// Condition to request disable send
      A #s_OPO98_Dispatch;// Correcting of the item is completed
      O #s_Request_Merge_Action;// Merge action is requested
      O #s_Transfer_Sort_Active;// Sorting a carrier is active
      O #s_Transfer_Merge_Active;
      O(;// When carrier at TRS01 is for OPO and TRS05 is not ready to receive an item
      A #t_TRS01_Item_Req_Sort;
      AN #s_TRS05_Ready_To_Receive;// TRS05 contain an item or not RTR
      );
      O #t_TRS05_Item_For_Merge;// Item is ready to be merged at the induct position
      O #s_TRS02_Req_Dis_Send;// Sorting is required for an item with valid LNK
      O #s_Merge_Act_Prst_PEC_Occ;// Merge action is active and the present PEC is still occupied
      = #t_TRS01_Ext_Req_Dis_Send;

      CALL #s_TRS01_FB_EQP_Basic
      (  i_ID_Section                := #i_TRS01_ID ,
         i_Basic_Offset              := #i_TRS01_Setting.Basic.Offset ,
         i_DB_PLT                    := #i_TRS01_DB_PLT ,
         i_DB_PLT_DwnStr             := #i_TRS02_DB_PLT ,
         i_DB_Event                  := "DB_Event_Section" ,
         i_Conveyor_Speed            := #s_TRS01_Selected_Speed ,
         i_Run_Out_Distance          := #s_TRS01_Selected_Run_Out ,
         i_Start_Up_Distance         := #s_TRS01_Selected_Startup ,
         i_Minimum_Gap               := #i_TRS01_Setting.Basic.Minimum_Gap ,
         i_Add_Gap_Stop              := #i_TRS01_Setting.Basic.Add_Gap_Stop ,
         i_Minimum_H2H               := #i_TRS01_Setting.Basic.Minimum_H2H ,
         i_Add_H2H_Stop              := #i_TRS01_Setting.Basic.Add_H2H_Stop ,
         i_CFG_Cascade_Delay_Time    := 30 ,
         i_CFG_Strt_Up_T_E_Save      := "DB_Setting".common.Start_Up_Time_E_Save ,
         i_CFG_Run_Out_E_Save        := "DB_Setting".common.Run_Out_Time_E_Save ,
         i_CFG_Stop_T_E_Save         := "DB_Setting".common.Stop_Time_E_Save ,
         i_PPI_Displacement          := 0 ,
         i_Dwnstr_PLT_Pos            := #s_TRS01_EOS_PEC_Pos ,
         i_CFG_Disbl_E_Save          := "DB_Setting".common.Disable_Energy_Saving ,
         i_CFG_Slave_Mode            := FALSE ,
         i_CFG_Del_Window_Codes      := FALSE ,
         i_Available_IO              := #i_IO_Available ,
         i_Safety_OK                 := #i_Safety_OK ,
         i_CMD_Enable                := #i_CMD_Enable ,
         i_CMD_Start                 := #i_CMD_Start ,
         i_Ext_Req_Stop              := #s_TRS01_Ext_Req_Stop ,
         i_Ext_Req_Halt              := FALSE ,
         i_Ext_Req_Dis_Send          := #t_TRS01_Ext_Req_Dis_Send ,
         i_Ext_Req_Rst_ESave         := FALSE ,
         i_OS_Direction_Change       := FALSE ,
         i_Clr_PLT_Data              := #s_TRS01_ST_LMS_Not_Auto ,
         o_External                  := #o_TRS01_Ext_Outputs ,
         o_Motor_Run                 := #s_TRS01_Motor_Run ,
         o_ST_Items                  := #o_TRS01_ST_Items ,
         o_ST_Running                := #o_TRS01_ST_Running ,
         o_ST_Started                := #o_TRS01_ST_Started ,
         o_ST_Request_Halt           := #o_TRS01_ST_Req_Halt ,
         o_ST_Request_Stop           := #o_TRS01_ST_Req_Stop ,
         o_ST_External_Stop          := #o_TRS01_ST_Ext_Stop ,
         o_Ready_To_Restart          := #s_TRS01_Ready_To_Restart
      );

      CALL #s_TRS01_FB_TRK_Track_EOS
      (  i_Setting                   := #i_TRS01_Setting.Tracking ,
         i_DB_PLT                    := #i_TRS01_DB_PLT ,
         i_Event_DB                  := "DB_Event_Section" ,
         i_Position_PEC_Update       := #s_TRS01_EOS_PEC_Pos ,
         i_LPOS                      := #s_TRS01_EOS_PEC_LPOS ,
         i_Length_Dif_Accepted       := 0 ,
         i_CFG_Num_Missing_Error     := 3 ,
         i_CFG_Upd_Perf_WN_Level     := 80 ,
         i_CFG_Weighing_Factor       := 10 ,
         i_CFG_Default_Record        := #i_CFG_Default_Record ,
         i_Trigger_Send_Stat         := #i_Send_Statistics ,
         i_CMD_Reset                 := #i_CMD_Reset ,
         i_CFG_Clear_Double_Data     := TRUE ,
         i_OS_Direction_Change       := FALSE ,
         i_HW_MTR_Not_Auto           := #s_TRS01_ST_LMS_Not_Auto ,
         o_ST_PEC_Miss               := #s_TRS01_ST_EOS_PEC_Miss ,
         o_ST_PEC_BadTrack           := #o_TRS01_ST_EOS_PEC_BadTr
      );

      AN "M_Hardware_PN";
      JCN HA01;

      CALL #s_TRS01_FB_HW_MltSpd_LMS
      (  i_CMD_Send_Stat             := #i_Send_Statistics ,
         i_DB_PLT                    := #i_TRS01_DB_PLT ,
         i_Event_DB                  := "DB_Event_Section" ,
         i_Speed1                    := #i_TRS01_Setting.Hardware.Speed1 ,
         i_Speed1_Run_Out_Dist       := #i_TRS01_Setting.Hardware.Speed1_Run_Out_Dist ,
         i_Speed1_Start_Up_Dist      := #i_TRS01_Setting.Hardware.Speed1_Start_Up_Dist ,
         i_CFG_Motor_Switch_Time     := 0 ,
         i_CMD_Select_Speed          := 1 ,
         i_Available_IO              := #i_IO_Available ,
         i_LMS_NotPrsnt              := #i_TRS01_LMS_Not_Prsnt ,
         i_LMS_Error                 := #i_TRS01_LMS_Error ,
         i_IO_LMS_Auto               := #i_TRS01_IO_LMS_Auto ,
         i_IO_LMS_Healthy            := #i_TRS01_IO_LMS_Healthy ,
         i_CMD_Reset                 := #i_CMD_Reset ,
         i_CMD_Req_Motor_Run         := #s_TRS01_Motor_Run ,
         o_IO_MTR_Fwd                := #o_TRS01_IO_MTR_Fwd ,
         o_IO_MTR_Rev                := #o_TRS01_IO_MTR_Rev ,
         o_IO_Speed_Select1          := #o_TRS01_IO_Speed_Select1 ,
         o_IO_Speed_Select2          := #o_TRS01_IO_Speed_Select2 ,
         o_ST_ASI_NotPrsnt           := #s_TRS01_ST_LMS_Not_Prsnt ,
         o_ST_ASI_Err                := #s_TRS01_ST_LMS_Error ,
         o_ST_LMS_Not_Auto           := #s_TRS01_ST_LMS_Not_Auto ,
         o_ST_LMS_Not_Hthy           := #s_TRS01_ST_LMS_Not_Hthy ,
         o_Select_Conveyor_Speed     := #s_TRS01_Selected_Speed ,
         o_Select_Run_Out_Dist       := #s_TRS01_Selected_Run_Out ,
         o_Select_Started_Up_Dist    := #s_TRS01_Selected_Startup
      );

      JU HA02;

HA01:      CALL #s_TRS01_FB_HW_MTR_PN_LMS
      (  i_CMD_Send_Stat             := #i_Send_Statistics ,
         i_DB_PLT                    := #i_TRS01_DB_PLT ,
         i_Event_DB                  := "DB_Event_Section" ,
         i_Speed                     := #i_TRS01_Setting.Hardware.Speed1 ,
         i_Run_Out_Dist              := #i_TRS01_Setting.Hardware.Speed1_Run_Out_Dist ,
         i_Start_Up_Dist             := #i_TRS01_Setting.Hardware.Speed1_Start_Up_Dist ,
         i_CFG_Motor_Switch_Time     := 0 ,
         i_CFG_In_Hardw_ID           := #i_TRS01_CFG_LMS_In_Hardw_ID ,
         i_CFG_Out_Hardw_ID          := #i_TRS01_CFG_LMS_Out_Hardw_ID ,
         i_Available_IO              := #i_IO_Available ,
         i_CMD_Reset                 := #i_CMD_Reset ,
         i_CMD_Req_Motor_Run         := #s_TRS01_Motor_Run ,
         o_ST_FieldB_NotPrsnt        := #s_TRS01_ST_LMS_Not_Prsnt ,
         o_ST_FieldB_Error           := #s_TRS01_ST_LMS_Error ,
         o_ST_LMS_Not_Auto           := #s_TRS01_ST_LMS_Not_Auto ,
         o_ST_LMS_Not_Hthy           := #s_TRS01_ST_LMS_Not_Hthy ,
         o_Select_Conveyor_Speed     := #s_TRS01_Selected_Speed ,
         o_Select_Run_Out_Dist       := #s_TRS01_Selected_Run_Out ,
         o_Select_Started_Up_Dist    := #s_TRS01_Selected_Startup
      );

HA02:      NOP 0;

      CALL #s_TRS01_FB_DAT_T
      (  i_ID                        := #i_TRS01_ID ,
         i_DB_Event                  := "DB_Event_Section" ,
         i_DB_PLT_Lost_And_Found     := #i_DB_PLT_Lost_And_Found ,
         i_DB_Send_FIFO_PNPN         := #i_DB_Send_FIFO_PNPN
      );

      CALL #s_TRS01_FB_DAT
      (  i_ID_Section                := #i_TRS01_ID ,
         i_DB_Event                  := "DB_Event_Section" ,
         i_PLC_Log_FIFO_DB           := "DB_LOG_Event_FIFO" ,
         i_CFG_BPI_Log_Level         := "DB_Setting".common.External_Log_Level ,
         i_CFG_PLC_Log_Level         := "DB_Setting".common.Internal_Log_Level ,
         i_CFG_PLC_Log_Route_Msgs    := FALSE ,
         i_CFG_PLC_LOG_BPI_Stat      := FALSE
      );

NETWORK
TITLE = IA: Transport section TRS02
      NOP 0;

// Condition to request stop
      A #s_TRS02_ST_LMS_Not_Prsnt;// LMS and PEC related errors
      O #s_TRS02_ST_LMS_Error;
      O #s_TRS02_ST_LMS_Not_Auto;
      O #s_TRS02_ST_LMS_Not_Hthy;
      O(;// SWS, MSO and TRS04 errors considered-
      A #s_SWS03_STM_Err;// when sorting is required for an item
      A #s_Sorting_Required;
      );
      O #s_TRS04_ST_Prsnt_PEC_Blk;// Present PEC blockage shall stop TRS02 at all times
      O(;// ASi slave errors of HAC PEC
      O #s_TRS04_ST_FieldB_Not_Prsnt;
      O #s_TRS04_ST_FieldB_Error;
      A #i_IO_Available;
      );
      = #s_TRS02_Ext_Req_Stop;

// Condition to request halt
      AN #s_SWS03_Req_Down;// Whenever SWS is requested to go down
      O(;
      A #s_TRS02_Carr_In_Pos;// When carrier is in position, sorting is required
      A #s_Sorting_Required;
      );
      O(;// Consider SWS related errors if not in down position
      A #s_SWS03_ST_LMS_Not_Prsnt;
      O #s_SWS03_ST_LMS_Error;
      O #s_SWS03_ST_LMS_Not_Auto;
      O #s_SWS03_ST_LMS_Not_Hthy;
      O #s_SWS03_ST_Move_TimeOut;
      O #s_SWS03_ST_PS_Double;
      AN #s_SWS03_ST_Down;
      );
      O(;// Consider MSO related errors if not in down position
      A #s_MSO99_ST_LMS_Not_Prsnt;
      O #s_MSO99_ST_LMS_Error;
      O #s_MSO99_ST_LMS_Not_Auto;
      O #s_MSO99_ST_LMS_Not_Hthy;
      O #s_MSO99_ST_Move_TimeOut;
      O #s_MSO99_ST_PS_Double;
      AN #s_MSO99_ST_Down;
      );
      O(;// When merge action is active, SWS is down
      A #s_Transfer_Merge_Active;// and the downstream is not RTR
      AN #t_TRS02_Dwnstr_RTR;
      A #i_SWS03_IO_PS_Down;
      );
      O #s_TRS04_ST_HAC_PEC_Blk;// ASi slave and PEC errors of HAC PEC
      O #s_TRS04_ST_FieldB_Not_Prsnt;
      O #s_TRS04_ST_FieldB_Error;
      O #s_TRS04_ST_SOS_PEC_Blk;// ASi slave and PEC errors of TRS04
      ON #s_TRS04_IO_Available_LMS;
      O(;// Latch the halt if stopped while merge is active
      A #s_Transfer_Merge_Active;
      O #s_TRS02_Ext_Req_Halt;
      A #i_CMD_Controlled_Stop;
      );
      O #s_Transfer_Merge_Active;// When merge action is active
      = #s_TRS02_Ext_Req_Halt;

// Condition to disable send
      A #i_CMD_Controlled_Stop;
      = #s_TRS02_Ext_Req_Dis_Send;

// Condition to reset Esave
      AN #i_TRS04_IO_NOT_Prsnt_PEC;
      = #t_TRS02_Ext_Req_Rst_Esav;

      CALL #s_TRS02_FB_EQP_Basic
      (  i_ID_Section                := #i_TRS02_ID ,
         i_Basic_Offset              := #i_TRS02_Setting.Basic.Offset ,
         i_DB_PLT                    := #i_TRS02_DB_PLT ,
         i_DB_PLT_DwnStr             := #i_DB_PLT_Dwnstr ,
         i_DB_Event                  := "DB_Event_Section" ,
         i_Conveyor_Speed            := #s_TRS02_Selected_Speed ,
         i_Run_Out_Distance          := #s_TRS02_Selected_Run_Out ,
         i_Start_Up_Distance         := #s_TRS02_Selected_Startup ,
         i_Minimum_Gap               := #i_TRS02_Setting.Basic.Minimum_Gap ,
         i_Add_Gap_Stop              := #i_TRS02_Setting.Basic.Add_Gap_Stop ,
         i_Minimum_H2H               := #i_TRS02_Setting.Basic.Minimum_H2H ,
         i_Add_H2H_Stop              := #i_TRS02_Setting.Basic.Add_H2H_Stop ,
         i_CFG_Dieback_Position      := #t_TRS02_CFG_MSO_Pos ,
         i_CFG_Cascade_Delay_Time    := 0 ,
         i_CFG_Strt_Up_T_E_Save      := "DB_Setting".common.Start_Up_Time_E_Save ,
         i_CFG_Run_Out_E_Save        := "DB_Setting".common.Run_Out_Time_E_Save ,
         i_CFG_Stop_T_E_Save         := "DB_Setting".common.Stop_Time_E_Save ,
         i_PPI_Displacement          := 0 ,
         i_Dwnstr_PLT_Pos            := #s_TRS04_SOS_PEC_Pos ,
         i_CFG_Disbl_E_Save          := "DB_Setting".common.Disable_Energy_Saving ,
         i_CFG_Slave_Mode            := FALSE ,
         i_CFG_Del_Window_Codes      := FALSE ,
         i_Available_IO              := #i_IO_Available ,
         i_Safety_OK                 := #i_Safety_OK ,
         i_CMD_Enable                := #i_CMD_Enable ,
         i_CMD_Start                 := #i_CMD_Start ,
         i_Ext_Req_Stop              := #s_TRS02_Ext_Req_Stop ,
         i_Ext_Req_Halt              := #s_TRS02_Ext_Req_Halt ,
         i_Ext_Req_Dis_Send          := #s_TRS02_Ext_Req_Dis_Send ,
         i_Ext_Req_Rst_ESave         := #t_TRS02_Ext_Req_Rst_Esav ,
         i_OS_Direction_Change       := FALSE ,
         i_Clr_PLT_Data              := FALSE ,
         o_External                  := #o_TRS02_Ext_Outputs ,
         o_Motor_Run                 := #s_TRS02_Motor_Run ,
         o_ST_Items                  := #s_TRS02_ST_Items ,
         o_ST_Running                := #o_TRS02_ST_Running ,
         o_ST_Started                := #o_TRS02_ST_Started ,
         o_ST_Request_Halt           := #o_TRS02_ST_Req_Halt ,
         o_ST_Request_Stop           := #o_TRS02_ST_Req_Stop ,
         o_ST_External_Stop          := #o_TRS02_ST_Ext_Stop ,
         o_Ready_To_Restart          := #s_TRS02_Ready_To_Restart
      );

      CALL #s_TRS02_FB_TRK_No_PEC
      (  i_DB_PLT                    := #i_TRS02_DB_PLT ,
         i_Event_DB                  := "DB_Event_Section" ,
         i_HW_MTR_Not_Auto           := #s_TRS02_ST_LMS_Not_Auto
      );

// Select speed
      AN #s_TRS02_Req_2nd_Speed;
      JCN IA01;

      L 1;
      T #t_TRS02_Select_Speed;
      JU IA02;

IA01:      L 2;
      T #t_TRS02_Select_Speed;

IA02:      AN "M_Hardware_PN";
      JCN IA03;

      CALL #s_TRS02_FB_HW_MltSpd_LMS
      (  i_CMD_Send_Stat             := #i_Send_Statistics ,
         i_DB_PLT                    := #i_TRS02_DB_PLT ,
         i_Event_DB                  := "DB_Event_Section" ,
         i_Speed1                    := #i_TRS02_Setting.Hardware.Speed1 ,
         i_Speed1_Run_Out_Dist       := #i_TRS02_Setting.Hardware.Speed1_Run_Out_Dist ,
         i_Speed1_Start_Up_Dist      := #i_TRS02_Setting.Hardware.Speed1_Start_Up_Dist ,
         i_Speed2                    := #i_TRS02_Setting.Hardware.Speed2 ,
         i_Speed2_Run_Out_Dist       := #i_TRS02_Setting.Hardware.Speed2_Run_Out_Dist ,
         i_Speed2_Start_Up_Dist      := #i_TRS02_Setting.Hardware.Speed2_Start_Up_Dist ,
         i_CFG_Motor_Switch_Time     := 0 ,
         i_CMD_Select_Speed          := #t_TRS02_Select_Speed ,
         i_Available_IO              := #i_IO_Available ,
         i_LMS_NotPrsnt              := #i_TRS02_LMS_Not_Prsnt ,
         i_LMS_Error                 := #i_TRS02_LMS_Error ,
         i_IO_LMS_Auto               := #i_TRS02_IO_LMS_Auto ,
         i_IO_LMS_Healthy            := #i_TRS02_IO_LMS_Healthy ,
         i_CMD_Reset                 := #i_CMD_Reset ,
         i_CMD_Req_Motor_Run         := #s_TRS02_Motor_Run ,
         i_CMD_Req_Motor_Reverse     := FALSE ,
         o_IO_MTR_Fwd                := #o_TRS02_IO_MTR_Fwd ,
         o_IO_MTR_Rev                := #o_TRS02_IO_MTR_Rev ,
         o_IO_Speed_Select1          := #o_TRS02_IO_Speed_Select1 ,
         o_IO_Speed_Select2          := #o_TRS02_IO_Speed_Select2 ,
         o_ST_ASI_NotPrsnt           := #s_TRS02_ST_LMS_Not_Prsnt ,
         o_ST_ASI_Err                := #s_TRS02_ST_LMS_Error ,
         o_ST_LMS_Not_Auto           := #s_TRS02_ST_LMS_Not_Auto ,
         o_ST_LMS_Not_Hthy           := #s_TRS02_ST_LMS_Not_Hthy ,
         o_Select_Conveyor_Speed     := #s_TRS02_Selected_Speed ,
         o_Select_Run_Out_Dist       := #s_TRS02_Selected_Run_Out ,
         o_Select_Started_Up_Dist    := #s_TRS02_Selected_Startup
      );

      JU IA04;

// By default use speed 1
IA03:      L #i_TRS02_Setting.Hardware.Speed1;
      T #t_TRS02_Speed;
      L #i_TRS02_Setting.Hardware.Speed1_Run_Out_Dist;
      T #t_TRS02_Run_Out_Dist;
      L #i_TRS02_Setting.Hardware.Speed1_Start_Up_Dist;
      T #t_TRS02_Start_Up_Dist;

// Determine if speed 2 is selected
      L #t_TRS02_Select_Speed;
      L 2;
      ==I;
      JCN IA05;

      L #i_TRS02_Setting.Hardware.Speed2;
      T #t_TRS02_Speed;
      L #i_TRS02_Setting.Hardware.Speed2_Run_Out_Dist;
      T #t_TRS02_Run_Out_Dist;
      L #i_TRS02_Setting.Hardware.Speed2_Start_Up_Dist;
      T #t_TRS02_Start_Up_Dist;

IA05:      CALL #s_TRS02_FB_HW_MTR_PN_LMS
      (  i_CMD_Send_Stat             := #i_Send_Statistics ,
         i_DB_PLT                    := #i_TRS02_DB_PLT ,
         i_Event_DB                  := "DB_Event_Section" ,
         i_Speed                     := #t_TRS02_Speed ,
         i_Run_Out_Dist              := #t_TRS02_Run_Out_Dist ,
         i_Start_Up_Dist             := #t_TRS02_Start_Up_Dist ,
         i_CFG_In_Hardw_ID           := #i_TRS02_CFG_LMS_In_Hardw_ID ,
         i_CFG_Out_Hardw_ID          := #i_TRS02_CFG_LMS_Out_Hardw_ID ,
         i_Available_IO              := #i_IO_Available ,
         i_CMD_Reset                 := #i_CMD_Reset ,
         i_CMD_Req_Motor_Run         := #s_TRS02_Motor_Run ,
         o_ST_FieldB_NotPrsnt        := #s_TRS02_ST_LMS_Not_Prsnt ,
         o_ST_FieldB_Error           := #s_TRS02_ST_LMS_Error ,
         o_ST_LMS_Not_Auto           := #s_TRS02_ST_LMS_Not_Auto ,
         o_ST_LMS_Not_Hthy           := #s_TRS02_ST_LMS_Not_Hthy ,
         o_Select_Conveyor_Speed     := #s_TRS02_Selected_Speed ,
         o_Select_Run_Out_Dist       := #s_TRS02_Selected_Run_Out ,
         o_Select_Started_Up_Dist    := #s_TRS02_Selected_Startup
      );

IA04:      NOP 0;

      CALL #s_TRS02_FB_DAT_T
      (  i_ID                        := #i_TRS02_ID ,
         i_DB_Event                  := "DB_Event_Section" ,
         i_DB_PLT_Lost_And_Found     := #i_DB_PLT_Lost_And_Found ,
         i_DB_Send_FIFO_PNPN         := #i_DB_Send_FIFO_PNPN
      );

      CALL #s_TRS02_FB_DAT
      (  i_ID_Section                := #i_TRS02_ID ,
         i_DB_Event                  := "DB_Event_Section" ,
         i_PLC_Log_FIFO_DB           := "DB_LOG_Event_FIFO" ,
         i_CFG_BPI_Log_Level         := "DB_Setting".common.External_Log_Level ,
         i_CFG_PLC_Log_Level         := "DB_Setting".common.Internal_Log_Level ,
         i_CFG_PLC_Log_Route_Msgs    := FALSE ,
         i_CFG_PLC_LOG_BPI_Stat      := FALSE
      );

NETWORK
TITLE = JA: Switch section SWS03 (TSS)
      NOP 0;

// SWS Up   = Direction A = Motor up
// SWS Down = Direction B = Motor Down
// Section up status
      A #i_IO_Available;
      A #i_SWS03_IO_PS_Up;
      AN #i_SWS03_IO_PS_Down;
      = #s_SWS03_ST_Up;

// Section down status
      A #i_IO_Available;
      A #i_SWS03_IO_PS_Down;
      AN #i_SWS03_IO_PS_Up;
      = #s_SWS03_ST_Down;

// Check for error transfer module
      A #s_SWS03_ST_LMS_Not_Prsnt;
      O #s_SWS03_ST_LMS_Error;
      O #s_SWS03_ST_LMS_Not_Auto;
      O #s_SWS03_ST_LMS_Not_Hthy;
      O #s_SWS03_ST_Move_TimeOut;
      O #s_SWS03_ST_PS_Double;
      O #s_TRS04_ST_LMS_Not_Prsnt;
      O #s_TRS04_ST_LMS_Error;
      O #s_TRS04_ST_LMS_Not_Auto;
      O #s_TRS04_ST_LMS_Not_Hthy;
      O #s_TRS04_ST_Prsnt_PEC_Blk;
      O #s_TRS04_ST_SOS_PEC_Blk;
      O #s_TRS04_ST_SOS_PEC_Miss;
      O #s_TRS04_ST_FieldB_Not_Prsnt;
      O #s_TRS04_ST_FieldB_Error;
      O #s_TRS04_ST_HAC_PEC_Blk;
      O #s_MSO99_ST_LMS_Not_Prsnt;
      O #s_MSO99_ST_LMS_Error;
      O #s_MSO99_ST_LMS_Not_Auto;
      O #s_MSO99_ST_LMS_Not_Hthy;
      O #s_MSO99_ST_Move_TimeOut;
      O #s_MSO99_ST_PS_Double;
      = #s_SWS03_STM_Err;

// Condition to request stop
      A #s_SWS03_STM_Err;
      = #s_SWS03_Ext_Req_Stop;

// Condition to request position up while sorting
      A #t_TRS02_Stopped;
      A #s_TRS02_Carr_In_Pos;
      AN #i_CMD_Controlled_Stop;
      O #s_Transfer_Sort_Active;
      = #t_SWS03_Req_Up_Sorting;

// Item in position on lift after merge
      A #s_TRS04_ST_Items;
      A #s_TRS04_ST_Started;
      AN #s_TRS04_ST_Running;
      AN #s_TRS05_ST_Items;
      A #i_TRS04_IO_NOT_HAC_PEC;
      AN #i_TRS04_IO_NOT_Prsnt_PEC;
      = #s_Carrier_On_Lift_Merge;

// Condition to request position up while merging
      A #s_Request_Merge_Action;
      O(;
      A #s_Transfer_Merge_Active;
      AN #s_Carrier_On_Lift_Merge;
      );
      = #t_SWS03_Req_Up_Merging;

// Condition to request position down
      AN #t_SWS03_Req_Up_Merging;
      AN #t_SWS03_Req_Up_Sorting;
      O(;
      A #i_CMD_Start;
      AN #s_SWS03_ST_Down;
      AN #s_Transfer_Sort_Active;
      AN #s_Request_Merge_Action;
      AN #s_Transfer_Merge_Active;
      );
      = #s_SWS03_Req_Down;

      CALL #s_SWS03_FB_EQP_Switch
      (  i_Available_IO              := #i_IO_Available ,
         i_Safety_OK                 := #i_Safety_OK ,
         i_CMD_Enable                := #i_CMD_Enable ,
         i_CMD_Start                 := #i_CMD_Start ,
         i_CMD_Reset                 := #i_CMD_Reset ,
         i_IO_PS_A                   := #i_SWS03_IO_PS_Up ,
         i_IO_PS_B                   := #i_SWS03_IO_PS_Down ,
         i_Ext_Req_Stop              := #s_SWS03_Ext_Req_Stop ,
         i_Ext_Req_Halt              := FALSE ,
         i_Req_Dir_B                 := #s_SWS03_Req_Down ,
         i_Timeout_Dir               := #i_SWS03_Setting.Timeout_Dir ,
         o_CMD_MTR_Run               := #s_SWS03_Motor_Run ,
         o_CMD_MTR_Reverse           := #s_SWS03_Motor_Reverse ,
         o_ST_Running                := #o_SWS03_ST_Running ,
         o_ST_Started                := #o_SWS03_ST_Started ,
         o_ST_Request_Halt           := #o_SWS03_ST_Req_Halt ,
         o_ST_Request_Stop           := #o_SWS03_ST_Req_Stop ,
         o_ST_External_Stop          := #o_SWS03_ST_Ext_Stop ,
         o_ST_Movement_Time_out      := #s_SWS03_ST_Move_TimeOut ,
         o_ST_PS_Double              := #s_SWS03_ST_PS_Double ,
         o_Ready_To_Restart          := #s_SWS03_Ready_To_Restart
      );

      AN "M_Hardware_PN";
      JCN JA01;

      CALL #s_SWS03_FB_HW_MTR_2D_LMS
      (  i_CMD_Send_Stat             := #i_Send_Statistics ,
         i_Event_DB                  := "DB_Event_Section" ,
         i_CFG_Motor_Switch_Time     := 0 ,
         i_Available_IO              := #i_IO_Available ,
         i_Quick_Stop                := TRUE ,
         i_LMS_NotPrsnt              := #i_SWS03_LMS_Not_Prsnt ,
         i_LMS_Error                 := #i_SWS03_LMS_Error ,
         i_IO_LMS_Auto               := #i_SWS03_IO_LMS_Auto ,
         i_IO_LMS_Healthy            := #i_SWS03_IO_LMS_Healthy ,
         i_CMD_Reset                 := #i_CMD_Reset ,
         i_CMD_Req_Motor_Run         := #s_SWS03_Motor_Run ,
         i_CMD_Req_Motor_Reverse     := #s_SWS03_Motor_Reverse ,
         o_IO_MTR_Fwd                := #o_SWS03_IO_MTR_Up ,
         o_IO_MTR_Rev                := #o_SWS03_IO_MTR_Down ,
         o_IO_MTR_Dis_Quick_Stop     := #o_SWS03_IO_Dis_QS ,
         o_ST_ASI_NotPrsnt           := #s_SWS03_ST_LMS_Not_Prsnt ,
         o_ST_ASI_Err                := #s_SWS03_ST_LMS_Error ,
         o_ST_LMS_Not_Auto           := #s_SWS03_ST_LMS_Not_Auto ,
         o_ST_LMS_Not_Hthy           := #s_SWS03_ST_LMS_Not_Hthy
      );

      JU JA02;

JA01:      CALL #s_SWS03_FB_HW_MTR_2D_PN_LMS
      (  i_CMD_Send_Stat             := #i_Send_Statistics ,
         i_Event_DB                  := "DB_Event_Section" ,
         i_CFG_Motor_Switch_Time     := 0 ,
         i_CFG_In_Hardw_ID           := #i_SWS03_CFG_LMS_In_Hardw_ID ,
         i_CFG_Out_Hardw_ID          := #i_SWS03_CFG_LMS_Out_Hardw_ID ,
         i_Available_IO              := #i_IO_Available ,
         i_CMD_Reset                 := #i_CMD_Reset ,
         i_CMD_Req_Motor_Run         := #s_SWS03_Motor_Run ,
         i_CMD_Req_Motor_Reverse     := #s_SWS03_Motor_Reverse ,
         o_ST_FieldB_NotPrsnt        := #s_SWS03_ST_LMS_Not_Prsnt ,
         o_ST_FieldB_Error           := #s_SWS03_ST_LMS_Error ,
         o_ST_LMS_Not_Auto           := #s_SWS03_ST_LMS_Not_Auto ,
         o_ST_LMS_Not_Hthy           := #s_SWS03_ST_LMS_Not_Hthy
      );

JA02:      NOP 0;

      CALL #s_SWS03_FB_DAT_T
      (  i_ID                        := #i_SWS03_ID ,
         i_DB_Event                  := "DB_Event_Section"
      );

      CALL #s_SWS03_FB_DAT
      (  i_ID_Section                := #i_SWS03_ID ,
         i_DB_Event                  := "DB_Event_Section" ,
         i_PLC_Log_FIFO_DB           := "DB_LOG_Event_FIFO" ,
         i_CFG_BPI_Log_Level         := "DB_Setting".common.External_Log_Level ,
         i_CFG_PLC_Log_Level         := "DB_Setting".common.Internal_Log_Level ,
         i_CFG_PLC_Log_Route_Msgs    := FALSE ,
         i_CFG_PLC_LOG_BPI_Stat      := FALSE
      );

NETWORK
TITLE = KA: Activate 2nd speed TRS04
//When a leading edge is found from a configurable point on TRS04, the TRS will
//switch to the 2nd speed. This is done to reduce the impact of the carrier
//against the side guarding.
      NOP 0;

      L #i_TRS04_CFG_2nd_Spd_Pos;
      L 30;// Add 30cm extra, to also find leading edge in END PLT (Dummy PLT)
      +I;
      T #t_Search_Window;

      CALL "FC_PLT_Srch_Inf_Dwn"
      (  i_DB_PLT_Num                := #t_TRS04_DB_PLT_Num ,
         i_Position                  := #i_TRS04_CFG_2nd_Spd_Pos ,
         i_Window                    := #t_Search_Window ,
         i_Info                      := 1 ,
         o_Position                  := #t_Not_Used_Int ,
         o_Info                      := #t_Not_Used_Int ,
         o_LNK                       := #t_Fnd_Link_2nd_Speed ,
         o_DB_PLT_Num                := #t_Not_Used_Int ,
         o_Number_Items_Found        := #t_Not_Used_Int
      );

// When a link has been found, switch to 2nd speed
      L #t_Fnd_Link_2nd_Speed;
      L 0;
      >I;
      A #s_Transfer_Merge_Active;
      JCN KA01;

      L 2;
      T #t_TRS04_Select_Speed;
      JU KA99;

KA01:      L 1;
      T #t_TRS04_Select_Speed;

KA99:      NOP 0;

NETWORK
TITLE = LA: Push carrier out of HAC PEC
//Push carrier out of the HAC PEC to avoid deadlock during transfer merge
      NOP 0;

      AN #i_TRS04_IO_NOT_HAC_PEC;
      A #t_TRS04_Operational;
      A #t_TRS04_Stopped;
      A #s_SWS03_ST_Up;
      A #s_Transfer_Merge_Active;
      = #t_Push_Carr_Timer_Start;

      CALL "FC_On_Dly_T_0.1s"
      (  i_Start                     := #t_Push_Carr_Timer_Start ,
         i_Enable_Dly                := TRUE ,
         i_Time_Value                := 45 ,
         i_Current_Value             := #s_Push_Carr_Timer_CV ,
         o_Status                    := #t_Push_Carr_Timer_Done ,
         o_Current_Value             := #s_Push_Carr_Timer_CV
      );

      OPN #i_TRS05_DB_PLT;
      A #t_Push_Carr_Timer_Start;
      JCN LA99;

      CLR;
      = %DBX10.6;// Item at handover

LA99:      NOP 0;

NETWORK
TITLE = MA: Transport section TRS04 (TTS)
//Note that the SOS PEC connects to the TRS04 LMS but is located on section 02
//not TRS04. The SOS PEC therefor updates the section 02 tracking.
      NOP 0;

      CALL #s_TRS04_FB_EQP_Switch_D
      (  i_DB_PLT                    := #i_TRS04_DB_PLT ,
         i_DB_PLT_UpStr              := #i_TRS04_DB_PLT_End ,
         i_DB_PLT_DwnStr             := #i_TRS05_DB_PLT ,
         i_CMD_Reverse               := #s_Req_Reverse_TRS05 ,
         i_CFG_Cascade_Delay_FWD     := 0 ,
         i_CFG_Cascade_Delay_REV     := 0 ,
         o_OS_Direction_Change       := #s_TRS04_OS_Dir_Change ,
         o_CMD_MTR_Reverse           := #s_TRS04_Motor_Reverse ,
         o_Cascade_Delay_Time        := #t_Not_Used_Int
      );

      AN #s_TRS04_Motor_Reverse;
      = #s_TRS04_Motor_Forward;

// IO Available for SOS and present PEC
      A #i_IO_Available;
      AN #s_TRS04_ST_LMS_Not_Prsnt;
      AN #s_TRS04_ST_LMS_Error;
      = #s_TRS04_IO_Available_LMS;

// Note the SOS PEC is located on the section 02, not TRS04
      CALL #s_TRS04_FB_EQP_PEC_SOS
      (  i_Setting                   := #i_TRS04_Setting.PEC_1 ,
         i_DB_PLT                    := #i_TRS02_DB_PLT ,
         i_DB_Event                  := "DB_Event_Section" ,
         i_Dwnstr_PLT_Pos            := 0 ,
         i_CFG_Blockage_Length       := #i_CFG_Blockage_Length_L ,
         i_CFG_Delay_On_Filter       := 15 ,
         i_CFG_Delay_Off_Filter      := 0 ,
         i_CFG_Flickering_Length     := 60 ,
         i_CFG_Min_Product_Length    := 60 ,
         i_CFG_Preset_PEC_Latch      := #s_TRS04_ST_LMS_Not_Auto ,
         i_CFG_Track_Present         := TRUE ,
         i_CFG_Reset_Block_PEC_Oc    := FALSE ,
         i_IO_NOT_PEC                := #i_TRS04_IO_NOT_SOS_PEC ,
         i_Eqp_Available_IO          := #s_TRS04_IO_Available_LMS ,
         i_CMD_Reset                 := #i_CMD_Reset ,
         o_LPOS                      := #s_TRS04_SOS_PEC_LPOS ,
         o_PEC_Position              := #s_TRS04_SOS_PEC_Pos ,
         o_ST_PEC_Blk                := #s_TRS04_ST_SOS_PEC_Blk
      );

// Determine if the present PEC is occupied during a merge action
      A #s_Transfer_Merge_Active;
      AN #i_TRS04_IO_NOT_Prsnt_PEC;
      S #s_Merge_Act_Prst_PEC_Occ;

      A #i_TRS04_IO_NOT_Prsnt_PEC;
      R #s_Merge_Act_Prst_PEC_Occ;

// Selection of displacement for present PEC blockage detection
      A #s_SWS03_ST_Up;
      JCN MA01;

      L #t_TRS04_Displ;// Displacement of transfer
      JU MA02;

MA01:      L #t_TRS02_Displ;// Displacement of mainline TB
MA02:      T #t_Displ_PECT_Prst;

// Blockage length present PEC
      L #i_CFG_Blockage_Length_L;
      L "DB_Setting".Common_TTT.SBT_Length;// Additional SBT length because of the (+/-)diagonal position of present PEC
      +I;
      T #t_PECT_Prst_Blck_length;// Blockage length present PEC

      CALL #s_TRS04_FB_EQP_PECT_Prst
      (  i_CFG_Blockage_Length       := #t_PECT_Prst_Blck_length ,
         i_CFG_Delay_On_Filter       := 0 ,
         i_CFG_Reset_Block_PEC_Oc    := FALSE ,
         i_CFG_Time_Displacement     := TRUE ,
         i_IO_NOT_PEC                := #i_TRS04_IO_NOT_Prsnt_PEC ,
         i_Eqp_Available_IO          := #s_TRS04_IO_Available_LMS ,
         i_CMD_Reset                 := #i_CMD_Reset ,
         i_Displacement              := #t_Displ_PECT_Prst ,
         o_ST_PEC_Blk                := #s_TRS04_ST_Prsnt_PEC_Blk ,
         o_PEC_Flap_Filter           := #s_TRS04_Prsnt_PEC_Latch
      );

// IO Available for HAC PEC
      A #i_IO_Available;
      AN #s_TRS04_ST_FieldB_Not_Prsnt;
      AN #s_TRS04_ST_FieldB_Error;
      = #t_TRS04_IO_Available_FieldB;

// Determine the displacement for the HAC PEC
// When running forward the displacement from TRS05 must be used
// When running reverse the displacement from TRS04 must be used
      A #s_TRS04_Motor_Forward;
      JCN MA03;

      L #t_TRS05_Displ;
      T #t_TRS04_HAC_PEC_Displ;// HAC PEC displacement when running forward
      JU MA04;

MA03:      L #t_TRS04_Displ;
      T #t_TRS04_HAC_PEC_Displ;// HAC PEC displacement when running reverse

MA04:      CALL #s_TRS04_FB_EQP_PECT_HAC
      (  i_CFG_Blockage_Length       := #i_CFG_Blockage_Length_W ,
         i_CFG_Delay_On_Filter       := 15 ,
         i_CFG_Reset_Block_PEC_Oc    := FALSE ,
         i_CFG_Time_Displacement     := TRUE ,
         i_IO_NOT_PEC                := #i_TRS04_IO_NOT_HAC_PEC ,
         i_Eqp_Available_IO          := #t_TRS04_IO_Available_FieldB ,
         i_CMD_Reset                 := #i_CMD_Reset ,
         i_Displacement              := #t_TRS04_HAC_PEC_Displ ,
         o_ST_PEC_Blk                := #s_TRS04_HAC_PEC_Blk ,
         o_PEC_Flap_Filter           := #s_TRS04_HAC_PEC_Latch
      );

// When the instance is downloaded and the HAC PEC is blocked, then make the PEC blockage
      AN #i_TRS04_IO_NOT_HAC_PEC;
      AN #s_Done;
      A #t_TRS04_IO_Available_FieldB;
      O #s_TRS04_HAC_PEC_Blk;
      O #t_Push_Carr_Timer_Done;
      S #s_TRS04_ST_HAC_PEC_Blk;

      A #i_TRS04_IO_NOT_HAC_PEC;
      A #i_CMD_Reset;
      R #s_TRS04_ST_HAC_PEC_Blk;

      AN "M_Hardware_PN";
      JCN MA05;

      CALL #s_TRS04_FB_HW_ASi
      (  i_Req_Output_1              := FALSE ,
         i_Req_Output_2              := FALSE ,
         i_Req_Output_3              := FALSE ,
         i_Req_Output_4              := FALSE ,
         i_CMD_Reset                 := #i_CMD_Reset ,
         i_Available_IO              := #i_IO_Available ,
         i_ASI_NotPrsnt              := #i_TRS04_ASI_Not_Prsnt ,
         i_Slave_Error               := #i_TRS04_ASI_Error ,
         i_CFG_Delay_Time            := 5 ,
         o_ST_ASI_NotPrsnt           := #s_TRS04_ST_ASI_Not_Prsnt ,
         o_ST_ASI_Error              := #s_TRS04_ST_ASI_Error
      );

      A #s_TRS04_ST_ASI_Not_Prsnt;
      = #s_TRS04_ST_FieldB_Not_Prsnt;
      A #s_TRS04_ST_ASI_Error;
      = #s_TRS04_ST_FieldB_Error;
      JU MA06;

MA05:      CALL #s_TRS04_FB_HW_Profinet
      (  i_Req_Output_1              := FALSE ,
         i_Req_Output_2              := FALSE ,
         i_Req_Output_3              := FALSE ,
         i_Req_Output_4              := FALSE ,
         i_CMD_Reset                 := #i_CMD_Reset ,
         i_Available_IO              := #i_IO_Available ,
         i_CFG_Hardw_ID              := #i_TRS04_CFG_Hardw_ID ,
         i_CFG_Delay_Time            := 0 ,
         o_ST_FieldB_NotPrsnt        := #s_TRS04_ST_FieldB_Not_Prsnt ,
         o_ST_FieldB_Error           := #s_TRS04_ST_FieldB_Error
      );

MA06:      NOP 0;

// Condition to request stop
      A #s_SWS03_STM_Err;
      = #s_TRS04_Ext_Req_Stop;

// Condition to request halt while merging
      A #s_OPO98_Dispatch;
      O #s_Request_Merge_Action;
      O(;
      AN #s_TRS05_ST_Started;
      A #s_Transfer_Merge_Active;
      );
      ON #s_SWS03_ST_Up;
      = #t_TRS04_Req_Halt_Merging;

// Condition to request halt while sorting
      ON #s_MSO99_ST_Down;
      O(;
      AN #s_TRS05_ST_Started;
      O #s_TRS05_ST_Items;
      AN #s_Transfer_Sort_Active;
      );
      A #s_Transfer_Sort_Active;
      = #t_TRS04_Req_Halt_Sorting;

// Condition to request halt
      A #t_TRS04_Req_Halt_Merging;
      O #t_TRS04_Req_Halt_Sorting;
      O #s_TRS04_Req_Halt;
      O(;// Item is ready to merge or TRS02 has items-
      A #t_TRS05_Item_For_Merge;// when downstream is not RTR
      O #s_TRS02_ST_Items;
      AN #t_TRS02_Dwnstr_RTR;
      );
      O(;// Latch the halt if stopped while merge is active
      A #s_Transfer_Merge_Active;
      O #s_TRS04_Ext_Req_Halt;
      A #i_SWS03_IO_PS_Down;
      A #i_CMD_Controlled_Stop;
      );
      ON #s_SWS03_ST_Up;
      ON #t_TRS02_Operational;
      = #s_TRS04_Ext_Req_Halt;

// Condition to request reset energy save
      A #s_TRS04_Prsnt_PEC_Latch;
      A #s_SWS03_ST_Up;
      = #t_TRS04_Ext_Req_Rst_ESav;

      CALL #s_TRS04_FB_EQP_Basic
      (  i_ID_Section                := #i_TRS04_ID ,
         i_Basic_Offset              := #i_TRS04_Setting.Basic.Offset ,
         i_DB_PLT                    := #i_TRS04_DB_PLT ,
         i_DB_PLT_DwnStr             := #i_TRS05_DB_PLT ,
         i_DB_Event                  := "DB_Event_Section" ,
         i_Conveyor_Speed            := #s_TRS04_Selected_Speed ,
         i_Run_Out_Distance          := #s_TRS04_Selected_Run_Out ,
         i_Start_Up_Distance         := #s_TRS04_Selected_Startup ,
         i_Minimum_Gap               := #i_TRS04_Setting.Basic.Minimum_Gap ,
         i_Add_Gap_Stop              := #i_TRS04_Setting.Basic.Add_Gap_Stop ,
         i_Minimum_H2H               := #i_TRS04_Setting.Basic.Minimum_H2H ,
         i_Add_H2H_Stop              := #i_TRS04_Setting.Basic.Add_H2H_Stop ,
         i_CFG_Cascade_Delay_Time    := 0 ,
         i_CFG_Strt_Up_T_E_Save      := "DB_Setting".common.Start_Up_Time_E_Save ,
         i_CFG_Run_Out_E_Save        := "DB_Setting".common.Run_Out_Time_E_Save ,
         i_CFG_Stop_T_E_Save         := "DB_Setting".common.Stop_Time_E_Save ,
         i_PPI_Displacement          := 0 ,
         i_Dwnstr_PLT_Pos            := 0 ,
         i_CFG_Disbl_E_Save          := "DB_Setting".common.Disable_Energy_Saving ,
         i_CFG_Slave_Mode            := FALSE ,
         i_CFG_Del_Window_Codes      := FALSE ,
         i_Available_IO              := #i_IO_Available ,
         i_Safety_OK                 := #i_Safety_OK ,
         i_CMD_Enable                := #i_CMD_Enable ,
         i_CMD_Start                 := #i_CMD_Start ,
         i_Ext_Req_Stop              := #s_TRS04_Ext_Req_Stop ,
         i_Ext_Req_Halt              := #s_TRS04_Ext_Req_Halt ,
         i_Ext_Req_Dis_Send          := FALSE ,
         i_Ext_Req_Rst_ESave         := #t_TRS04_Ext_Req_Rst_ESav ,
         i_OS_Direction_Change       := #s_TRS04_OS_Dir_Change ,
         i_Clr_PLT_Data              := FALSE ,
         o_External                  := #o_TRS04_Ext_Outputs ,
         o_Motor_Run                 := #s_TRS04_Motor_Run ,
         o_ST_Items                  := #s_TRS04_ST_Items ,
         o_ST_Running                := #s_TRS04_ST_Running ,
         o_ST_Started                := #s_TRS04_ST_Started ,
         o_ST_Request_Halt           := #o_TRS04_ST_Req_Halt ,
         o_ST_Request_Stop           := #o_TRS04_ST_Req_Stop ,
         o_ST_External_Stop          := #o_TRS04_ST_Ext_Stop ,
         o_Ready_To_Restart          := #s_TRS04_Ready_To_Restart
      );

// Conditions for motor run
      A #s_TRS04_Motor_Run;
      O #t_Push_Carr_Timer_Start;
      = #t_TRS04_Motor_Run;

      CALL #s_TRS04_FB_TRK_Track_SOS
      (  i_Setting                   := #i_TRS04_Setting.Tracking ,
         i_DB_PLT                    := #i_TRS02_DB_PLT ,
         i_Event_DB                  := "DB_Event_Section" ,
         i_Position_PEC_Update       := #s_TRS04_SOS_PEC_Pos ,
         i_LPOS                      := #s_TRS04_SOS_PEC_LPOS ,
         i_Length_Dif_Accepted       := 0 ,
         i_CFG_Num_Missing_Error     := 3 ,
         i_CFG_Upd_Perf_WN_Level     := 80 ,
         i_CFG_Weighing_Factor       := 10 ,
         i_CFG_Default_Record        := #i_CFG_Default_Record ,
         i_Trigger_Send_Stat         := #i_Send_Statistics ,
         i_CMD_Reset                 := #i_CMD_Reset ,
         i_CFG_Clear_Double_Data     := TRUE ,
         i_OS_Direction_Change       := FALSE ,
         i_HW_MTR_Not_Auto           := #s_TRS04_ST_LMS_Not_Auto ,
         o_ST_PEC_Miss               := #s_TRS04_ST_SOS_PEC_Miss ,
         o_ST_PEC_BadTrack           := #o_TRS04_ST_SOS_PEC_BadTr
      );

      AN "M_Hardware_PN";
      JCN MA07;

      CALL #s_TRS04_FB_HW_MltSpd_LMS
      (  i_CMD_Send_Stat             := #i_Send_Statistics ,
         i_DB_PLT                    := #i_TRS04_DB_PLT ,
         i_Event_DB                  := "DB_Event_Section" ,
         i_Speed1                    := #i_TRS04_Setting.Hardware.Speed1 ,
         i_Speed1_Run_Out_Dist       := #i_TRS04_Setting.Hardware.Speed1_Run_Out_Dist ,
         i_Speed1_Start_Up_Dist      := #i_TRS04_Setting.Hardware.Speed1_Start_Up_Dist ,
         i_Speed2                    := #i_TRS04_Setting.Hardware.Speed2 ,
         i_Speed2_Run_Out_Dist       := #i_TRS04_Setting.Hardware.Speed2_Run_Out_Dist ,
         i_Speed2_Start_Up_Dist      := #i_TRS04_Setting.Hardware.Speed2_Start_Up_Dist ,
         i_CFG_Motor_Switch_Time     := 300 ,
         i_CMD_Select_Speed          := #t_TRS04_Select_Speed ,
         i_Available_IO              := #i_IO_Available ,
         i_LMS_NotPrsnt              := #i_TRS04_LMS_Not_Prsnt ,
         i_LMS_Error                 := #i_TRS04_LMS_Error ,
         i_IO_LMS_Auto               := #i_TRS04_IO_LMS_Auto ,
         i_IO_LMS_Healthy            := #i_TRS04_IO_LMS_Healthy ,
         i_CMD_Reset                 := #i_CMD_Reset ,
         i_CMD_Req_Motor_Run         := #t_TRS04_Motor_Run ,
         i_CMD_Req_Motor_Reverse     := #s_TRS04_Motor_Reverse ,
         o_IO_MTR_Fwd                := #o_TRS04_IO_MTR_Fwd ,
         o_IO_MTR_Rev                := #o_TRS04_IO_MTR_Rev ,
         o_IO_Speed_Select1          := #o_TRS04_IO_Speed_Select1 ,
         o_IO_Speed_Select2          := #o_TRS04_IO_Speed_Select2 ,
         o_ST_ASI_NotPrsnt           := #s_TRS04_ST_LMS_Not_Prsnt ,
         o_ST_ASI_Err                := #s_TRS04_ST_LMS_Error ,
         o_ST_LMS_Not_Auto           := #s_TRS04_ST_LMS_Not_Auto ,
         o_ST_LMS_Not_Hthy           := #s_TRS04_ST_LMS_Not_Hthy ,
         o_Select_Conveyor_Speed     := #s_TRS04_Selected_Speed ,
         o_Select_Run_Out_Dist       := #s_TRS04_Selected_Run_Out ,
         o_Select_Started_Up_Dist    := #s_TRS04_Selected_Startup ,
         o_Req_Halt                  := #s_TRS04_Req_Halt
      );

      JU MA08;

// By default use speed 1
MA07:      L #i_TRS04_Setting.Hardware.Speed1;
      T #t_TRS04_Speed;
      L #i_TRS04_Setting.Hardware.Speed1_Run_Out_Dist;
      T #t_TRS04_Run_Out_Dist;
      L #i_TRS04_Setting.Hardware.Speed1_Start_Up_Dist;
      T #t_TRS04_Start_Up_Dist;

// Determine if speed 2 is selected
      L #t_TRS04_Select_Speed;
      L 2;
      ==I;
      JCN MA09;

      L #i_TRS04_Setting.Hardware.Speed2;
      T #t_TRS04_Speed;
      L #i_TRS04_Setting.Hardware.Speed2_Run_Out_Dist;
      T #t_TRS04_Run_Out_Dist;
      L #i_TRS04_Setting.Hardware.Speed2_Start_Up_Dist;
      T #t_TRS04_Start_Up_Dist;

MA09:      CALL #s_TRS04_FB_HW_MTR_PN_LMS
      (  i_CMD_Send_Stat             := #i_Send_Statistics ,
         i_DB_PLT                    := #i_TRS04_DB_PLT ,
         i_Event_DB                  := "DB_Event_Section" ,
         i_Speed                     := #t_TRS04_Speed ,
         i_Run_Out_Dist              := #t_TRS04_Run_Out_Dist ,
         i_Start_Up_Dist             := #t_TRS04_Start_Up_Dist ,
         i_CFG_Motor_Switch_Time     := 300 ,
         i_CFG_In_Hardw_ID           := #i_TRS04_CFG_LMS_In_Hardw_ID ,
         i_CFG_Out_Hardw_ID          := #i_TRS04_CFG_LMS_Out_Hardw_ID ,
         i_Available_IO              := #i_IO_Available ,
         i_CMD_Reset                 := #i_CMD_Reset ,
         i_CMD_Req_Motor_Run         := #s_TRS04_Motor_Run ,
         i_CMD_Req_Motor_Reverse     := #s_TRS04_Motor_Reverse ,
         o_ST_FieldB_NotPrsnt        := #s_TRS04_ST_LMS_Not_Prsnt ,
         o_ST_FieldB_Error           := #s_TRS04_ST_LMS_Error ,
         o_ST_LMS_Not_Auto           := #s_TRS04_ST_LMS_Not_Auto ,
         o_ST_LMS_Not_Hthy           := #s_TRS04_ST_LMS_Not_Hthy ,
         o_Select_Conveyor_Speed     := #s_TRS04_Selected_Speed ,
         o_Select_Run_Out_Dist       := #s_TRS04_Selected_Run_Out ,
         o_Select_Started_Up_Dist    := #s_TRS04_Selected_Startup ,
         o_Req_Halt                  := #s_TRS04_Req_Halt
      );

MA08:      NOP 0;

      CALL #s_TRS04_FB_DAT_T
      (  i_ID                        := #i_TRS04_ID ,
         i_DB_Event                  := "DB_Event_Section" ,
         i_DB_PLT_Lost_And_Found     := #i_DB_PLT_Lost_And_Found ,
         i_DB_Send_FIFO_PNPN         := #i_DB_Send_FIFO_PNPN
      );

      CALL #s_TRS04_FB_DAT
      (  i_ID_Section                := #i_TRS04_ID ,
         i_DB_Event                  := "DB_Event_Section" ,
         i_PLC_Log_FIFO_DB           := "DB_LOG_Event_FIFO" ,
         i_CFG_BPI_Log_Level         := "DB_Setting".common.External_Log_Level ,
         i_CFG_PLC_Log_Level         := "DB_Setting".common.Internal_Log_Level ,
         i_CFG_PLC_Log_Route_Msgs    := FALSE ,
         i_CFG_PLC_LOG_BPI_Stat      := FALSE
      );

NETWORK
TITLE = NA: Mechanical stop object MSO99
      NOP 0;

// MSO Up   = Direction A = Motor up
// MSO Down = Direction B = Motor Down
// Section up status
      A #i_IO_Available;
      A #i_MSO99_IO_PS_Up;
      AN #i_MSO99_IO_PS_Down;
      = #o_MSO99_ST_Up;

// Section down status
      A #i_IO_Available;
      A #i_MSO99_IO_PS_Down;
      AN #i_MSO99_IO_PS_Up;
      = #s_MSO99_ST_Down;

// Request MSO99 to go up
      L #t_TRS02_Fnd_Items_Lead;
      L 0;
      >I;
      A #s_DP_Dir_Side;
      AN #s_Transfer_Sort_Active;
      A #s_TRS02_ST_Items;
      A #i_CMD_Enable;
      S #s_MSO99_Req_Up;

      A #s_DP_Dir_Straight;
      ON #s_TRS02_ST_Items;
      O #i_SWS03_IO_PS_Up;
      A #i_MSO99_IO_PS_Up;
      R #s_MSO99_Req_Up;

// Condition to request stop
      A #s_MSO99_ST_LMS_Not_Prsnt;
      O #s_MSO99_ST_LMS_Error;
      O #s_MSO99_ST_LMS_Not_Auto;
      O #s_MSO99_ST_LMS_Not_Hthy;
      O #s_MSO99_ST_Move_TimeOut;
      O #s_MSO99_ST_PS_Double;
      = #s_MSO99_Ext_Req_Stop;

// Condition to request position down
      AN #s_MSO99_Req_Up;
      = #s_MSO99_Req_Down;

      CALL #s_MSO99_FB_EQP_Switch
      (  i_Available_IO              := #i_IO_Available ,
         i_Safety_OK                 := #i_Safety_OK ,
         i_CMD_Enable                := #i_CMD_Enable ,
         i_CMD_Start                 := #i_CMD_Start ,
         i_CMD_Reset                 := #i_CMD_Reset ,
         i_IO_PS_A                   := #i_MSO99_IO_PS_Up ,
         i_IO_PS_B                   := #i_MSO99_IO_PS_Down ,
         i_Ext_Req_Stop              := #s_MSO99_Ext_Req_Stop ,
         i_Req_Dir_B                 := #s_MSO99_Req_Down ,
         i_Timeout_Dir               := #i_MSO99_Setting.Timeout_Dir ,
         o_CMD_MTR_Run               := #s_MSO99_Motor_Run ,
         o_CMD_MTR_Reverse           := #s_MSO99_Motor_Reverse ,
         o_ST_Running                := #o_MSO99_ST_Running ,
         o_ST_Started                := #o_MSO99_ST_Started ,
         o_ST_Request_Halt           := #o_MSO99_ST_Req_Halt ,
         o_ST_Request_Stop           := #o_MSO99_ST_Req_Stop ,
         o_ST_External_Stop          := #o_MSO99_ST_Ext_Stop ,
         o_ST_Movement_Time_out      := #s_MSO99_ST_Move_TimeOut ,
         o_ST_PS_Double              := #s_MSO99_ST_PS_Double ,
         o_Ready_To_Restart          := #s_MSO99_Ready_To_Restart
      );

      AN "M_Hardware_PN";
      JCN NA01;

      CALL #s_MSO99_FB_HW_MTR_2D_LMS
      (  i_CMD_Send_Stat             := #i_Send_Statistics ,
         i_Event_DB                  := "DB_Event_Section" ,
         i_CFG_Motor_Switch_Time     := 0 ,
         i_Available_IO              := #i_IO_Available ,
         i_Quick_Stop                := TRUE ,
         i_LMS_NotPrsnt              := #i_MSO99_LMS_Not_Prsnt ,
         i_LMS_Error                 := #i_MSO99_LMS_Error ,
         i_IO_LMS_Auto               := #i_MSO99_IO_LMS_Auto ,
         i_IO_LMS_Healthy            := #i_MSO99_IO_LMS_Healthy ,
         i_CMD_Reset                 := #i_CMD_Reset ,
         i_CMD_Req_Motor_Run         := #s_MSO99_Motor_Run ,
         i_CMD_Req_Motor_Reverse     := #s_MSO99_Motor_Reverse ,
         o_IO_MTR_Fwd                := #o_MSO99_IO_MTR_Up ,
         o_IO_MTR_Rev                := #o_MSO99_IO_MTR_Down ,
         o_IO_MTR_Dis_Quick_Stop     := #o_MSO99_IO_Dis_QS ,
         o_ST_ASI_NotPrsnt           := #s_MSO99_ST_LMS_Not_Prsnt ,
         o_ST_ASI_Err                := #s_MSO99_ST_LMS_Error ,
         o_ST_LMS_Not_Auto           := #s_MSO99_ST_LMS_Not_Auto ,
         o_ST_LMS_Not_Hthy           := #s_MSO99_ST_LMS_Not_Hthy
      );

      JU NA02;

NA01:      CALL #s_MSO99_FB_HW_MTR_2D_PN_LMS
      (  i_CMD_Send_Stat             := #i_Send_Statistics ,
         i_Event_DB                  := "DB_Event_Section" ,
         i_CFG_Motor_Switch_Time     := 0 ,
         i_CFG_In_Hardw_ID           := #i_MSO99_CFG_LMS_In_Hardw_ID ,
         i_CFG_Out_Hardw_ID          := #i_MSO99_CFG_LMS_Out_Hardw_ID ,
         i_Available_IO              := #i_IO_Available ,
         i_CMD_Reset                 := #i_CMD_Reset ,
         i_CMD_Req_Motor_Run         := #s_MSO99_Motor_Run ,
         i_CMD_Req_Motor_Reverse     := #s_MSO99_Motor_Reverse ,
         o_ST_FieldB_NotPrsnt        := #s_MSO99_ST_LMS_Not_Prsnt ,
         o_ST_FieldB_Error           := #s_MSO99_ST_LMS_Error ,
         o_ST_LMS_Not_Auto           := #s_MSO99_ST_LMS_Not_Auto ,
         o_ST_LMS_Not_Hthy           := #s_MSO99_ST_LMS_Not_Hthy
      );

NA02:      NOP 0;

      CALL #s_MSO99_FB_DAT_T
      (  i_ID                        := #i_MSO99_ID ,
         i_DB_Event                  := "DB_Event_Section"
      );

      CALL #s_MSO99_FB_DAT
      (  i_ID_Section                := #i_MSO99_ID ,
         i_DB_Event                  := "DB_Event_Section" ,
         i_PLC_Log_FIFO_DB           := "DB_LOG_Event_FIFO" ,
         i_CFG_BPI_Log_Level         := "DB_Setting".common.External_Log_Level ,
         i_CFG_PLC_Log_Level         := "DB_Setting".common.Internal_Log_Level ,
         i_CFG_PLC_Log_Route_Msgs    := FALSE ,
         i_CFG_PLC_LOG_BPI_Stat      := FALSE
      );

NETWORK
TITLE = OA: Transport section TRS05
      NOP 0;

      CALL #s_TRS05_FB_EQP_Switch_D
      (  i_DB_PLT                    := #i_TRS05_DB_PLT ,
         i_DB_PLT_UpStr              := #i_TRS04_DB_PLT ,
         i_DB_PLT_DwnStr             := #i_TRS05_DB_PLT_End ,
         i_CMD_Reverse               := #s_Req_Reverse_TRS05 ,
         i_CFG_Cascade_Delay_FWD     := 0 ,
         i_CFG_Cascade_Delay_REV     := 0 ,
         o_OS_Direction_Change       := #s_TRS05_OS_Dir_Change ,
         o_CMD_MTR_Reverse           := #s_TRS05_Motor_Reverse
      );

      AN #s_TRS05_Motor_Reverse;
      = #s_TRS05_Motor_Forward;

      A(;
      A #s_TRS05_Motor_Forward;
      A #t_TRS05_Req_2nd_Spd;
      );
      O(;
      A #s_OPO98_Dispatch;
      AN #s_TRS05_Item_At_Dieback;
      );
      = #s_TRS05_Req_2nd_Speed;

      A #i_IO_Available;
      AN #s_TRS05_ST_LMS_Not_Prsnt;
      AN #s_TRS05_ST_LMS_Error;
      = #t_TRS05_IO_Available;

      CALL #s_TRS05_FB_EQP_PEC2D_SOS
      (  i_Setting                   := #i_TRS05_Setting.PEC_2 ,
         i_DB_PLT                    := #i_TRS05_DB_PLT ,
         i_DB_Event                  := "DB_Event_Section" ,
         i_Dwnstr_PLT_Pos            := 0 ,
         i_CFG_Blockage_Length       := #i_CFG_Blockage_Length_W ,
         i_CFG_Delay_On_Filter       := 10 ,
         i_CFG_Delay_Off_Filter      := 0 ,
         i_CFG_Flickering_Length     := 45 ,
         i_CFG_Min_Product_Length    := 45 ,
         i_CFG_Track_Present         := TRUE ,
         i_CFG_Reset_Block_PEC_Oc    := FALSE ,
         i_IO_NOT_PEC                := #i_TRS05_IO_NOT_SOS_PEC ,
         i_CFG_Preset_PEC_Latch      := FALSE ,
         i_Eqp_Available_IO          := #t_TRS05_IO_Available ,
         i_CMD_Reset                 := #i_CMD_Reset ,
         i_Disable_Update_Funct      := #s_TRS05_Motor_Forward ,
         o_LPOS                      := #s_TRS05_SOS_PEC_LPOS ,
         o_PEC_Position              := #s_TRS05_SOS_PEC_Pos ,
         o_ST_PEC_Blk                := #s_TRS05_ST_SOS_PEC_Blk
      );

      CALL #s_TRS05_FB_EQP_PEC2D_EOS
      (  i_Setting                   := #i_TRS05_Setting.PEC_1 ,
         i_DB_PLT                    := #i_TRS05_DB_PLT ,
         i_DB_Event                  := "DB_Event_Section" ,
         i_Dwnstr_PLT_Pos            := 0 ,
         i_CFG_Blockage_Length       := #i_CFG_Blockage_Length_W ,
         i_CFG_Delay_On_Filter       := 15 ,
         i_CFG_Delay_Off_Filter      := 0 ,
         i_CFG_Flickering_Length     := 25 , //45 inasaw jfk#3709
         i_CFG_Min_Product_Length    := 45 ,
         i_CFG_Track_Present         := TRUE ,
         i_CFG_Reset_Block_PEC_Oc    := FALSE ,
         i_IO_NOT_PEC                := #i_TRS05_IO_NOT_EOS_PEC ,
         i_CFG_Preset_PEC_Latch      := FALSE ,
         i_Eqp_Available_IO          := #t_TRS05_IO_Available ,
         i_CMD_Reset                 := #i_CMD_Reset ,
         i_Disable_Update_Funct      := #s_TRS05_Motor_Reverse ,
         o_LPOS                      := #s_TRS05_EOS_PEC_LPOS ,
         o_PEC_Position              := #s_TRS05_EOS_PEC_Pos ,
         o_ST_PEC_Blk                := #s_TRS05_ST_EOS_PEC_Blk
      );

// Set PEC position and basic offset depending on running forward or reverse
      A #s_TRS05_Motor_Forward;
      JCN OA01;

      L #s_TRS05_EOS_PEC_Pos;
      T #s_TRS05_PEC_Pos;

      L #i_TRS05_Setting.Basic_FWD.Offset;
      T #t_TRS05_Setting.Offset;

      L #i_TRS05_Setting.Basic_FWD.Minimum_Gap;
      T #t_TRS05_Setting.Minimum_Gap;

      L #i_TRS05_Setting.Basic_FWD.Add_Gap_Stop;
      T #t_TRS05_Setting.Add_Gap_Stop;

      L #i_TRS05_Setting.Basic_FWD.Minimum_H2H;
      T #t_TRS05_Setting.Minimum_H2H;

      L #i_TRS05_Setting.Basic_FWD.Add_H2H_Stop;
      T #t_TRS05_Setting.Add_H2H_Stop;

      JU OA02;

OA01:      L #s_TRS05_SOS_PEC_Pos;
      T #s_TRS05_PEC_Pos;

      L #i_TRS05_Setting.Basic_REV.Offset;
      T #t_TRS05_Setting.Offset;

      L #i_TRS05_Setting.Basic_REV.Minimum_Gap;
      T #t_TRS05_Setting.Minimum_Gap;

      L #i_TRS05_Setting.Basic_REV.Add_Gap_Stop;
      T #t_TRS05_Setting.Add_Gap_Stop;

      L #i_TRS05_Setting.Basic_REV.Minimum_H2H;
      T #t_TRS05_Setting.Minimum_H2H;

      L #i_TRS05_Setting.Basic_REV.Add_H2H_Stop;
      T #t_TRS05_Setting.Add_H2H_Stop;

// Condition to request stop
OA02:      A #s_SWS03_STM_Err;
      O #s_TRS05_ST_LMS_Not_Prsnt;
      O #s_TRS05_ST_LMS_Error;
      O #s_TRS05_ST_LMS_Not_Auto;
      O #s_TRS05_ST_LMS_Not_Hthy;
      O #s_TRS05_ST_EOS_PEC_Blk;
      O #s_TRS05_ST_EOS_PEC_Miss;
      O #s_TRS05_ST_SOS_PEC_Blk;
      O #s_TRS05_ST_SOS_PEC_Miss;
      = #s_TRS05_Ext_Req_Stop;

// Condition to request halt
// Motor reverse signal is implemented in s_TRS05_Item_At_Dieback
      AN #t_TRS04_Motor_On_Speed;// TRS04 is not on speed and item at dieback pos
      A #s_TRS05_Item_At_Dieback;
      O #s_TRS05_Req_Halt;// OR Request halt from HW layer
      O #i_TRS05_Ext_Req_Halt;
      = #s_TRS05_Ext_Req_Halt;

      CALL #s_TRS05_FB_EQP_Basic
      (  i_ID_Section                := #i_TRS05_ID ,
         i_Basic_Offset              := #t_TRS05_Setting.Offset ,
         i_DB_PLT                    := #i_TRS05_DB_PLT ,
         i_DB_PLT_DwnStr             := #i_TRS05_DB_PLT_End ,
         i_DB_Event                  := "DB_Event_Section" ,
         i_Conveyor_Speed            := #s_TRS05_Selected_Speed ,
         i_Run_Out_Distance          := #s_TRS05_Selected_Run_Out ,
         i_Start_Up_Distance         := #s_TRS05_Selected_Startup ,
         i_Minimum_Gap               := #t_TRS05_Setting.Minimum_Gap ,
         i_Add_Gap_Stop              := #t_TRS05_Setting.Add_Gap_Stop ,
         i_Minimum_H2H               := #t_TRS05_Setting.Minimum_H2H ,
         i_Add_H2H_Stop              := #t_TRS05_Setting.Add_H2H_Stop ,
         i_CFG_Cascade_Delay_Time    := 0 ,
         i_CFG_Strt_Up_T_E_Save      := "DB_Setting".common.Start_Up_Time_E_Save ,
         i_CFG_Run_Out_E_Save        := "DB_Setting".common.Run_Out_Time_E_Save ,
         i_CFG_Stop_T_E_Save         := "DB_Setting".common.Stop_Time_E_Save ,
         i_PPI_Displacement          := 0 ,
         i_Dwnstr_PLT_Pos            := #s_TRS05_PEC_Pos ,
         i_CFG_Disbl_E_Save          := "DB_Setting".common.Disable_Energy_Saving ,
         i_CFG_Slave_Mode            := FALSE ,
         i_CFG_Del_Window_Codes      := FALSE ,
         i_Available_IO              := #i_IO_Available ,
         i_Safety_OK                 := #i_Safety_OK ,
         i_CMD_Enable                := #i_CMD_Enable ,
         i_CMD_Start                 := #i_CMD_Start ,
         i_Ext_Req_Stop              := #s_TRS05_Ext_Req_Stop ,
         i_Ext_Req_Halt              := #s_TRS05_Ext_Req_Halt ,
         i_Ext_Req_Dis_Send          := FALSE ,
         i_Ext_Req_Rst_ESave         := FALSE ,
         i_OS_Direction_Change       := #s_TRS05_OS_Dir_Change ,
         i_Clr_PLT_Data              := FALSE ,
         o_External                  := #o_TRS05_Ext_Outputs ,
         o_Motor_Run                 := #s_TRS05_Motor_Run ,
         o_ST_Items                  := #s_TRS05_ST_Items ,
         o_ST_Running                := #o_TRS05_ST_Running ,
         o_ST_Started                := #s_TRS05_ST_Started ,
         o_ST_Request_Halt           := #o_TRS05_ST_Req_Halt ,
         o_ST_Request_Stop           := #o_TRS05_ST_Req_Stop ,
         o_ST_External_Stop          := #o_TRS05_ST_Ext_Stop ,
         o_Ready_To_Restart          := #s_TRS05_Ready_To_Restart
      );

// If running in forward direction
      CALL #s_TRS05_FB_TRK_Track_EOS
      (  i_Setting                   := #i_TRS05_Setting.Tracking_FWD ,
         i_DB_PLT                    := #i_TRS05_DB_PLT ,
         i_Event_DB                  := "DB_Event_Section" ,
         i_Position_PEC_Update       := #s_TRS05_EOS_PEC_Pos ,
         i_LPOS                      := #s_TRS05_EOS_PEC_LPOS ,
         i_Length_Dif_Accepted       := 0 ,
         i_CFG_Num_Missing_Error     := 3 ,
         i_CFG_Upd_Perf_WN_Level     := 80 ,
         i_CFG_Weighing_Factor       := 10 ,
         i_CFG_Default_Record        := #i_CFG_Default_Record ,
         i_Trigger_Send_Stat         := #i_Send_Statistics ,
         i_CMD_Reset                 := #i_CMD_Reset ,
         i_CFG_Clear_Double_Data     := TRUE ,
         i_OS_Direction_Change       := FALSE ,
         i_HW_MTR_Not_Auto           := #s_TRS05_ST_LMS_Not_Auto ,
         i_Disable_Update_Funct      := #s_TRS05_Motor_Reverse ,
         o_ST_PEC_Miss               := #s_TRS05_ST_EOS_PEC_Miss ,
         o_ST_PEC_BadTrack           := #o_TRS05_ST_EOS_PEC_BadTr
      );

// If running in reverse direction
      CALL #s_TRS05_FB_TRK_Track_SOS
      (  i_Setting                   := #i_TRS05_Setting.Tracking_REV ,
         i_DB_PLT                    := #i_TRS05_DB_PLT ,
         i_Event_DB                  := "DB_Event_Section" ,
         i_Position_PEC_Update       := #s_TRS05_SOS_PEC_Pos ,
         i_LPOS                      := #s_TRS05_SOS_PEC_LPOS ,
         i_Length_Dif_Accepted       := 0 ,
         i_CFG_Num_Missing_Error     := 3 ,
         i_CFG_Upd_Perf_WN_Level     := 80 ,
         i_CFG_Weighing_Factor       := 10 ,
         i_CFG_Default_Record        := #i_CFG_Default_Record ,
         i_Trigger_Send_Stat         := #i_Send_Statistics ,
         i_CMD_Reset                 := #i_CMD_Reset ,
         i_CFG_Clear_Double_Data     := TRUE ,
         i_OS_Direction_Change       := FALSE ,
         i_HW_MTR_Not_Auto           := #s_TRS05_ST_LMS_Not_Auto ,
         i_Disable_Update_Funct      := #s_TRS05_Motor_Forward ,
         o_ST_PEC_Miss               := #s_TRS05_ST_SOS_PEC_Miss ,
         o_ST_PEC_BadTrack           := #o_TRS05_ST_SOS_PEC_BadTr
      );

// Select speed
      AN #s_TRS05_Req_2nd_Speed;
      JCN OA03;

      L 1;
      T #t_TRS05_Select_Speed;
      JU OA04;

OA03:      L 2;
      T #t_TRS05_Select_Speed;

OA04:      AN "M_Hardware_PN";
      JCN OA05;

      CALL #s_TRS05_FB_HW_MltSpd_LMS
      (  i_CMD_Send_Stat             := #i_Send_Statistics ,
         i_DB_PLT                    := #i_TRS05_DB_PLT ,
         i_Event_DB                  := "DB_Event_Section" ,
         i_Speed1                    := #i_TRS05_Setting.Hardware.Speed1 ,
         i_Speed1_Run_Out_Dist       := #i_TRS05_Setting.Hardware.Speed1_Run_Out_Dist ,
         i_Speed1_Start_Up_Dist      := #i_TRS05_Setting.Hardware.Speed1_Start_Up_Dist ,
         i_Speed2                    := #i_TRS05_Setting.Hardware.Speed2 ,
         i_Speed2_Run_Out_Dist       := #i_TRS05_Setting.Hardware.Speed2_Run_Out_Dist ,
         i_Speed2_Start_Up_Dist      := #i_TRS05_Setting.Hardware.Speed2_Start_Up_Dist ,
         i_CFG_Motor_Switch_Time     := 300 ,
         i_CMD_Select_Speed          := #t_TRS05_Select_Speed ,
         i_Available_IO              := #i_IO_Available ,
         i_LMS_NotPrsnt              := #i_TRS05_LMS_Not_Prsnt ,
         i_LMS_Error                 := #i_TRS05_LMS_Error ,
         i_IO_LMS_Auto               := #i_TRS05_IO_LMS_Auto ,
         i_IO_LMS_Healthy            := #i_TRS05_IO_LMS_Healthy ,
         i_CMD_Reset                 := #i_CMD_Reset ,
         i_CMD_Req_Motor_Run         := #s_TRS05_Motor_Run ,
         i_CMD_Req_Motor_Reverse     := #s_TRS05_Motor_Reverse ,
         o_IO_MTR_Fwd                := #o_TRS05_IO_MTR_Fwd ,
         o_IO_MTR_Rev                := #o_TRS05_IO_MTR_Rev ,
         o_IO_Speed_Select1          := #o_TRS05_IO_Speed_Select1 ,
         o_IO_Speed_Select2          := #o_TRS05_IO_Speed_Select2 ,
         o_ST_ASI_NotPrsnt           := #s_TRS05_ST_LMS_Not_Prsnt ,
         o_ST_ASI_Err                := #s_TRS05_ST_LMS_Error ,
         o_ST_LMS_Not_Auto           := #s_TRS05_ST_LMS_Not_Auto ,
         o_ST_LMS_Not_Hthy           := #s_TRS05_ST_LMS_Not_Hthy ,
         o_Select_Conveyor_Speed     := #s_TRS05_Selected_Speed ,
         o_Select_Run_Out_Dist       := #s_TRS05_Selected_Run_Out ,
         o_Select_Started_Up_Dist    := #s_TRS05_Selected_Startup ,
         o_Req_Halt                  := #s_TRS05_Req_Halt
      );

      JU OA06;

// By default use speed 1
OA05:      L #i_TRS05_Setting.Hardware.Speed1;
      T #t_TRS05_Speed;
      L #i_TRS05_Setting.Hardware.Speed1_Run_Out_Dist;
      T #t_TRS05_Run_Out_Dist;
      L #i_TRS05_Setting.Hardware.Speed1_Start_Up_Dist;
      T #t_TRS05_Start_Up_Dist;

// Determine if speed 2 is selected
      L #t_TRS05_Select_Speed;
      L 2;
      ==I;
      JCN OA07;

      L #i_TRS05_Setting.Hardware.Speed2;
      T #t_TRS05_Speed;
      L #i_TRS05_Setting.Hardware.Speed2_Run_Out_Dist;
      T #t_TRS05_Run_Out_Dist;
      L #i_TRS05_Setting.Hardware.Speed2_Start_Up_Dist;
      T #t_TRS05_Start_Up_Dist;

OA07:      CALL #s_TRS05_FB_HW_MTR_PN_LMS
      (  i_CMD_Send_Stat             := #i_Send_Statistics ,
         i_DB_PLT                    := #i_TRS05_DB_PLT ,
         i_Event_DB                  := "DB_Event_Section" ,
         i_Speed                     := #t_TRS05_Speed ,
         i_Run_Out_Dist              := #t_TRS05_Run_Out_Dist ,
         i_Start_Up_Dist             := #t_TRS05_Start_Up_Dist ,
         i_CFG_Motor_Switch_Time     := 300 ,
         i_CFG_In_Hardw_ID           := #i_TRS05_CFG_LMS_In_Hardw_ID ,
         i_CFG_Out_Hardw_ID          := #i_TRS05_CFG_LMS_Out_Hardw_ID ,
         i_Available_IO              := #i_IO_Available ,
         i_CMD_Reset                 := #i_CMD_Reset ,
         i_CMD_Req_Motor_Run         := #s_TRS05_Motor_Run ,
         i_CMD_Req_Motor_Reverse     := #s_TRS05_Motor_Reverse ,
         o_ST_FieldB_NotPrsnt        := #s_TRS05_ST_LMS_Not_Prsnt ,
         o_ST_FieldB_Error           := #s_TRS05_ST_LMS_Error ,
         o_ST_LMS_Not_Auto           := #s_TRS05_ST_LMS_Not_Auto ,
         o_ST_LMS_Not_Hthy           := #s_TRS05_ST_LMS_Not_Hthy ,
         o_Select_Conveyor_Speed     := #s_TRS05_Selected_Speed ,
         o_Select_Run_Out_Dist       := #s_TRS05_Selected_Run_Out ,
         o_Select_Started_Up_Dist    := #s_TRS05_Selected_Startup ,
         o_Req_Halt                  := #s_TRS05_Req_Halt
      );

OA06:      NOP 0;

      CALL #s_TRS05_FB_DAT_T
      (  i_ID                        := #i_TRS05_ID ,
         i_DB_Event                  := "DB_Event_Section" ,
         i_DB_PLT_Lost_And_Found     := #i_DB_PLT_Lost_And_Found ,
         i_DB_Send_FIFO_PNPN         := #i_DB_Send_FIFO_PNPN
      );

      CALL #s_TRS05_FB_DAT
      (  i_ID_Section                := #i_TRS05_ID ,
         i_DB_Event                  := "DB_Event_Section" ,
         i_PLC_Log_FIFO_DB           := "DB_LOG_Event_FIFO" ,
         i_CFG_BPI_Log_Level         := "DB_Setting".common.External_Log_Level ,
         i_CFG_PLC_Log_Level         := "DB_Setting".common.Internal_Log_Level ,
         i_CFG_PLC_Log_Route_Msgs    := FALSE ,
         i_CFG_PLC_LOG_BPI_Stat      := FALSE
      );

NETWORK
TITLE = PA: Clear DB PLT of TRS02
// When the LMS is put in the NOT automatic mode the DB PLT will be cleared.
// This is done to make sure carriers that are removed from the transport section
// are also removed from the DB PLT in exceptional situations.
      NOP 0;

// Clear DB PLT when LMS is not automatic
      A #s_TRS02_ST_LMS_Not_Auto;
      A #i_TRS04_IO_NOT_Prsnt_PEC;
      = #t_TRS02_Clear_DB_PLT;

      CALL "FC_PLT_Clr_DB"
      (  i_Enable_Clr                := #t_TRS02_Clear_DB_PLT ,
         i_DB_PLT_Num                := #t_TRS02_DB_PLT_Num ,
         i_DB_Event_Num              := #t_DB_Event_Zone_Num
      );

// Clear item at handover signal in DB PLT when DB PLT is cleared
      OPN DB[ #t_TRS02_DB_PLT_Num];
      A #t_TRS02_Clear_DB_PLT;
      R %DBX10.6;// Item at handover position

NETWORK
TITLE = QA: Clear DB PLT of TRS04
//When the LMS is put in the NOT automatic mode the DB PLT will be cleared.
//This is done to make sure carriers that are removed from the transport section
//are also removed from the DB PLT in exceptional situations.
      NOP 0;

// Clear DB PLT when LMS is not automatic
      A #s_TRS04_ST_LMS_Not_Auto;
      A #i_TRS04_IO_NOT_Prsnt_PEC;
      = #t_TRS04_Clear_DB_PLT;

      CALL "FC_PLT_Clr_DB"
      (  i_Enable_Clr                := #t_TRS04_Clear_DB_PLT ,
         i_DB_PLT_Num                := #t_TRS04_DB_PLT_Num ,
         i_DB_Event_Num              := #t_DB_Event_Zone_Num
      );

// Clear item at handover signal in DB PLT when DB PLT is cleared
      OPN DB[ #t_TRS04_DB_PLT_Num];
      A #t_TRS04_Clear_DB_PLT;
      R %DBX10.6;// Item at handover position
      R #s_Transfer_Sort_Active;
      R #s_Transfer_Merge_Active;

NETWORK
TITLE = RA: Clear DB PLT of TRS05
// When the LMS is put in the NOT automatic mode the DB PLT will be cleared.
// This is done to make sure carriers that are removed from the transport section
// are also removed from the DB PLT in exceptional situations
      NOP 0;

// Clear DB PLT when LMS is not automatic
      A #s_TRS05_ST_LMS_Not_Auto;
      A #i_TRS05_IO_NOT_SOS_PEC;
      A #i_TRS05_IO_NOT_EOS_PEC;
      = #t_TRS05_Clear_DB_PLT;

      CALL "FC_PLT_Clr_DB"
      (  i_Enable_Clr                := #t_TRS05_Clear_DB_PLT ,
         i_DB_PLT_Num                := #t_TRS05_DB_PLT_Num ,
         i_DB_Event_Num              := #t_DB_Event_Zone_Num
      );

// Clear item at handover signal in DB PLT when DB PLT is cleared
      OPN DB[ #t_TRS05_DB_PLT_Num];
      A #t_TRS05_Clear_DB_PLT;
      R %DBX10.6;// Item at handover position

NETWORK
TITLE = SA: Write carrier in DB PLT of TRS02
//To make sure the carrier present on the transport section is also recognized in
//exceptional situations (for instance after download of a DB PLT or manual
//intervention) the carrier that is present on the transport section will be
//written into the DB PLT after this situation has been recovered.
//
//NOTE: This network needs to be positioned after the equipment network of the
//transport section where the leading and trailing edge will be written in. This
//is required because the done bit in the DB PLT is used to determine when the
//action is executed.
      NOP 0;

// Trigger negative flank of LMS not auto for writing PLT data (LMS back to automatic)
      A #s_TRS02_ST_LMS_Not_Auto;
      FN #s_TRS02_FN_Copy_LMS_Auto;
      = #s_TRS02_FN_ST_LMS_Auto;

// Write carrier into DB PLT of TRS when DB PLT is downloaded or LMS is put
// back into automatic mode and present PEC is still occupied
      A #s_TRS02_FN_ST_LMS_Auto;
      O #t_TRS02_FP_Done;
      AN #i_TRS04_IO_NOT_Prsnt_PEC;
      JCN SA99;

// Create new link number with correct default record
      CALL "FC_Gen_Default_LNK"
      (  i_LNK                       := 0 ,
         i_Default_Record            := #i_CFG_Default_Record ,
         i_DB_Event_Num              := #t_DB_Event_Zone_Num ,
         o_LNK                       := #t_Fnd_Link
      );

      L #t_Fnd_Link;
      L 0;
      >I;
      JCN SA99;

// Write leading edge in transport section
      CALL "FC_PLT_Write"
      (  i_DB_PLT_Num                := #t_TRS02_DB_PLT_Num ,
         i_Position                  := #t_TRS02_CFG_MSO_Pos ,
         i_Info_State                := WORD#16#0000 ,
         i_Info_Physical             := 1 ,
         i_LNK                       := #t_Fnd_Link ,
         i_DB_Event_Num              := #t_DB_Event_Zone_Num
      );

// Calculate position to write trailing edge
      L #t_TRS02_CFG_MSO_Pos;
      L #t_Carr_Length;
      +I;
      T #t_Write_Pos_Trailing;

// Write trailing edge in transport section
      CALL "FC_PLT_Write"
      (  i_DB_PLT_Num                := #t_TRS02_DB_PLT_Num ,
         i_Position                  := #t_Write_Pos_Trailing ,
         i_Info_State                := WORD#16#0000 ,
         i_Info_Physical             := 2 ,
         i_LNK                       := 0 ,
         i_DB_Event_Num              := #t_DB_Event_Zone_Num
      );

// Write DB PLT number to LNK record
      CALL "FC_Write_Int_Record"
      (  i_Record_Number             := #t_Fnd_Link ,
         i_P_INT_Record              := "DB_UDT_LNK_Record".DB_PLT_Number ,
         i_DB                        := "DB_LNK_List" ,
         i_INT                       := #t_TRS02_DB_PLT_Num ,
         i_DB_Event_Num              := #t_DB_Event_Zone_Num
      );

SA99:      NOP 0;

NETWORK
TITLE = SB: Write carrier in DB PLT of TRS04
//To make sure the carrier present on the transport section is also recognized in
//exceptional situations (for instance after download of a DB PLT or manual
//intervention) the carrier that is present on the transport section will be
//written into the DB PLT after this situation has been recovered.
//
//NOTE: This network needs to be positioned after the equipment network of the
//transport section where the leading and trailing edge will be written in. This
//is required because the done bit in the DB PLT is used to determine when the
//action is executed.
      NOP 0;

// Trigger negative flank of LMS not auto for writing PLT data (LMS back to automatic)
      A #s_TRS04_ST_LMS_Not_Auto;
      FN #s_TRS04_FN_Copy_LMS_Auto;
      = #s_TRS04_FN_ST_LMS_Auto;

// Write carrier into DB PLT of TRS when DB PLT is downloaded or LMS is put
// back into automatic mode and present PEC is still occupied
      A #s_TRS04_FN_ST_LMS_Auto;
      ON #s_Done;
      A #t_TRS04_Done;
      O #t_TRS04_FP_Done;
      AN #i_TRS04_IO_NOT_Prsnt_PEC;
      AN #s_SWS03_ST_Down;
      A #i_TRS04_IO_NOT_HAC_PEC;
      AN #t_TRS05_Item_At_HO;
      JCN SB01;

// Create new link number with correct default record
      CALL "FC_Gen_Default_LNK"
      (  i_LNK                       := 0 ,
         i_Default_Record            := #i_CFG_Default_Record ,
         i_DB_Event_Num              := #t_DB_Event_Zone_Num ,
         o_LNK                       := #t_Fnd_Link
      );

      L #t_Fnd_Link;
      L 0;
      >I;
      JCN SB99;

// Write leading edge in transport section
      CALL "FC_PLT_Write"
      (  i_DB_PLT_Num                := #t_TRS04_DB_PLT_Num ,
         i_Position                  := 0 ,
         i_Info_State                := WORD#16#0000 ,
         i_Info_Physical             := 1 ,
         i_LNK                       := #t_Fnd_Link ,
         i_DB_Event_Num              := #t_DB_Event_Zone_Num
      );

// Write trailing edge in transport section
      CALL "FC_PLT_Write"
      (  i_DB_PLT_Num                := #t_TRS04_DB_PLT_Num ,
         i_Position                  := #t_Carr_Width ,
         i_Info_State                := WORD#16#0000 ,
         i_Info_Physical             := 2 ,
         i_LNK                       := 0 ,
         i_DB_Event_Num              := #t_DB_Event_Zone_Num
      );

// Write DB PLT number to LNK record
      CALL "FC_Write_Int_Record"
      (  i_Record_Number             := #t_Fnd_Link ,
         i_P_INT_Record              := "DB_UDT_LNK_Record".DB_PLT_Number ,
         i_DB                        := "DB_LNK_List" ,
         i_INT                       := #t_TRS04_DB_PLT_Num ,
         i_DB_Event_Num              := #t_DB_Event_Zone_Num
      );

// Write carrier into DB PLT of TRS when DB PLT is downloaded or LMS is put
// back into automatic mode when handover from section 05 was busy
// s_LNK = 0 means that section 04 already handed over its leading edge
SB01:      A #s_TRS04_FN_ST_LMS_Auto;
      ON #s_Done;
      A #t_TRS04_Done;
      O #t_TRS04_FP_Done;
      A #s_SWS03_ST_Up;
      A #t_TRS05_Item_At_HO;
      A #s_Transfer_Merge_Active;
      A(;
      L #s_LNK;
      L 0;
      ==I;
      );
      JCN SB99;

// Create new link number with correct default record
      CALL "FC_Gen_Default_LNK"
      (  i_LNK                       := 0 ,
         i_Default_Record            := #i_CFG_Default_Record ,
         i_DB_Event_Num              := #t_DB_Event_Zone_Num ,
         o_LNK                       := #t_Fnd_Link
      );

      L #t_Fnd_Link;
      L 0;
      >I;
      JCN SB99;

// Write leading edge in transport section
      CALL "FC_PLT_Write"
      (  i_DB_PLT_Num                := #t_TRS04_DB_PLT_Num ,
         i_Position                  := 100 ,
         i_Info_State                := WORD#16#0000 ,
         i_Info_Physical             := 1 ,
         i_LNK                       := #t_Fnd_Link ,
         i_DB_Event_Num              := #t_DB_Event_Zone_Num
      );

// Write DB PLT number to LNK record
      CALL "FC_Write_Int_Record"
      (  i_Record_Number             := #t_Fnd_Link ,
         i_P_INT_Record              := "DB_UDT_LNK_Record".DB_PLT_Number ,
         i_DB                        := "DB_LNK_List" ,
         i_INT                       := #t_TRS04_DB_PLT_Num ,
         i_DB_Event_Num              := #t_DB_Event_Zone_Num
      );

SB99:      NOP 0;

NETWORK
TITLE = SC: Write carrier in DB PLT of TRS05
//To make sure the carrier present on the transport section is also recognized in
//exceptional situations (for instance after download of a DB PLT or manual
//intervention) the carrier that is present on the transport section will be
//written into the DB PLT after this situation has been recovered.
//
//NOTE: This network needs to be positioned after the equipment network of the
//transport section where the leading and trailing edge will be written in. This
//is required because the done bit in the DB PLT is used to determine when the
//action is executed.
      NOP 0;

// Trigger negative flank of LMS not auto for writing PLT data (LMS back to automatic)
      A #s_TRS05_ST_LMS_Not_Auto;
      FN #s_TRS05_FN_Copy_LMS_Auto;
      = #s_TRS05_FN_ST_LMS_Auto;

// Write carrier into DB PLT of TRS when DB PLT is downloaded or LMS is put
// back into automatic mode and PEC is still occupied
      A #s_TRS05_FN_ST_LMS_Auto;
      O #t_TRS05_FP_Done;
      ON #s_Done;
      AN #s_TRS05_ST_Items;
      A(;
      ON #i_TRS05_IO_NOT_SOS_PEC;
      ON #i_TRS05_IO_NOT_EOS_PEC;
      );
      JCN SC99;

// Create new link number with correct default record
      CALL "FC_Gen_Default_LNK"
      (  i_LNK                       := 0 ,
         i_Default_Record            := #i_CFG_Default_Record ,
         i_DB_Event_Num              := #t_DB_Event_Zone_Num ,
         o_LNK                       := #t_Fnd_Link
      );

      L #t_Fnd_Link;
      L 0;
      >I;
      JCN SC99;

      AN #i_TRS05_IO_NOT_EOS_PEC;
      JCN SC01;

      L 1;
      T #t_TRS05_Write_Position;
      JU SC02;

SC01:      AN #i_TRS05_IO_NOT_SOS_PEC;
      JCN SC02;

      L 65;
      T #t_TRS05_Write_Position;

// Write leading edge in transport section
SC02:      CALL "FC_PLT_Write"
      (  i_DB_PLT_Num                := #t_TRS05_DB_PLT_Num ,
         i_Position                  := #t_TRS05_Write_Position ,
         i_Info_State                := WORD#16#0000 ,
         i_Info_Physical             := 1 ,
         i_LNK                       := #t_Fnd_Link ,
         i_DB_Event_Num              := #t_DB_Event_Zone_Num
      );

// Calculate position to write trailing edge
      L #t_TRS05_Write_Position;// The position where the front of the carrier is located
      L #t_Carr_Width;
      +I;
      T #t_Write_Pos_Trailing;

// Write trailing edge in transport section
      CALL "FC_PLT_Write"
      (  i_DB_PLT_Num                := #t_TRS05_DB_PLT_Num ,
         i_Position                  := #t_Write_Pos_Trailing ,
         i_Info_State                := WORD#16#0000 ,
         i_Info_Physical             := 2 ,
         i_LNK                       := 0 ,
         i_DB_Event_Num              := #t_DB_Event_Zone_Num
      );

// Write DB PLT number to LNK record
      CALL "FC_Write_Int_Record"
      (  i_Record_Number             := #t_Fnd_Link ,
         i_P_INT_Record              := "DB_UDT_LNK_Record".DB_PLT_Number ,
         i_DB                        := "DB_LNK_List" ,
         i_INT                       := #t_TRS05_DB_PLT_Num ,
         i_DB_Event_Num              := #t_DB_Event_Zone_Num
      );

// Reset sequence for this item
      SET;
      R #s_Request_Merge_Action;
      R #s_Transfer_Merge_Active;
      R #s_Sorting_Required;
      R #s_Transfer_Sort_Active;

SC99:      NOP 0;

NETWORK
TITLE = TA: Send zone events
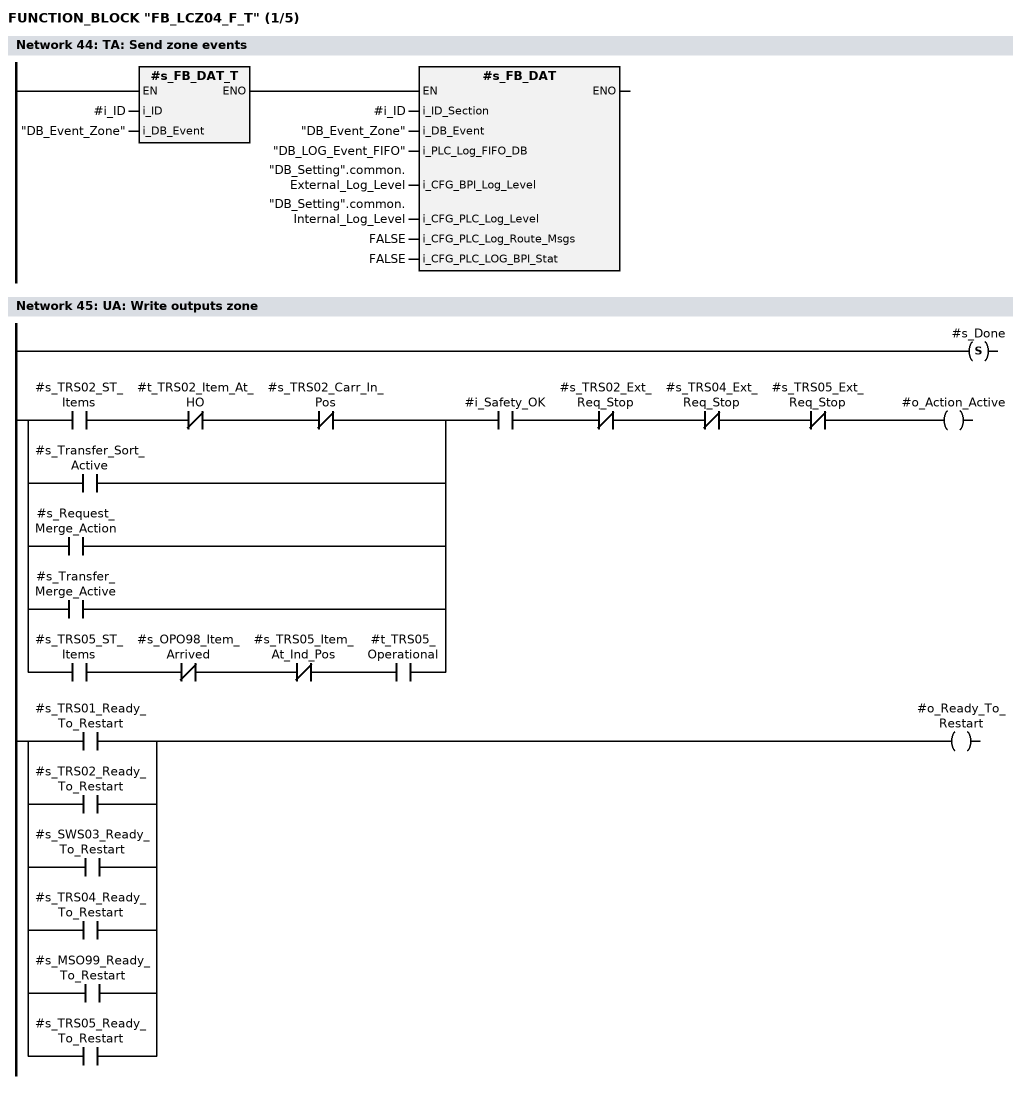
      NOP 0;

      CALL #s_FB_DAT_T
      (  i_ID                        := #i_ID ,
         i_DB_Event                  := "DB_Event_Zone"
      );

      CALL #s_FB_DAT
      (  i_ID_Section                := #i_ID ,
         i_DB_Event                  := "DB_Event_Zone" ,
         i_PLC_Log_FIFO_DB           := "DB_LOG_Event_FIFO" ,
         i_CFG_BPI_Log_Level         := "DB_Setting".common.External_Log_Level ,
         i_CFG_PLC_Log_Level         := "DB_Setting".common.Internal_Log_Level ,
         i_CFG_PLC_Log_Route_Msgs    := FALSE ,
         i_CFG_PLC_LOG_BPI_Stat      := FALSE
      );

NETWORK
TITLE = UA: Write outputs zone
      NOP 0;

// Set done bit indication (first scan finished)
      SET;
      S #s_Done;

// Action active
      O(;
      A #s_TRS02_ST_Items;
      AN #t_TRS02_Item_At_HO;
      AN #s_TRS02_Carr_In_Pos;
      );
      O #s_Transfer_Sort_Active;
      O #s_Request_Merge_Action;
      O #s_Transfer_Merge_Active;
      O(;
      A #s_TRS05_ST_Items;
      AN #s_OPO98_Item_Arrived;
      AN #s_TRS05_Item_At_Ind_Pos;
      A #t_TRS05_Operational;
      );
      A #i_Safety_OK;
      AN #s_TRS02_Ext_Req_Stop;
      AN #s_TRS04_Ext_Req_Stop;
      AN #s_TRS05_Ext_Req_Stop;
      = #o_Action_Active;

// Ready to restart
      A #s_TRS01_Ready_To_Restart;
      O #s_TRS02_Ready_To_Restart;
      O #s_SWS03_Ready_To_Restart;
      O #s_TRS04_Ready_To_Restart;
      O #s_MSO99_Ready_To_Restart;
      O #s_TRS05_Ready_To_Restart;
      = #o_Ready_To_Restart;

NETWORK
TITLE = VA: Write outputs TRS01
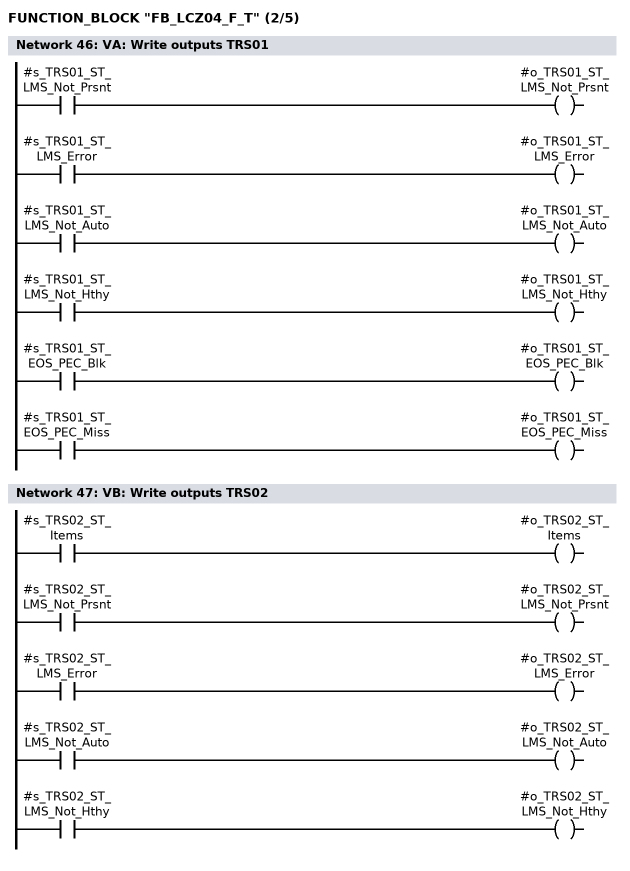
      NOP 0;

// Transfer static values to outputs
      A #s_TRS01_ST_LMS_Not_Prsnt;
      = #o_TRS01_ST_LMS_Not_Prsnt;
      A #s_TRS01_ST_LMS_Error;
      = #o_TRS01_ST_LMS_Error;
      A #s_TRS01_ST_LMS_Not_Auto;
      = #o_TRS01_ST_LMS_Not_Auto;
      A #s_TRS01_ST_LMS_Not_Hthy;
      = #o_TRS01_ST_LMS_Not_Hthy;
      A #s_TRS01_ST_EOS_PEC_Blk;
      = #o_TRS01_ST_EOS_PEC_Blk;
      A #s_TRS01_ST_EOS_PEC_Miss;
      = #o_TRS01_ST_EOS_PEC_Miss;

NETWORK
TITLE = VB: Write outputs TRS02
      NOP 0;

// Transfer static values to outputs
      A #s_TRS02_ST_Items;
      = #o_TRS02_ST_Items;
      A #s_TRS02_ST_LMS_Not_Prsnt;
      = #o_TRS02_ST_LMS_Not_Prsnt;
      A #s_TRS02_ST_LMS_Error;
      = #o_TRS02_ST_LMS_Error;
      A #s_TRS02_ST_LMS_Not_Auto;
      = #o_TRS02_ST_LMS_Not_Auto;
      A #s_TRS02_ST_LMS_Not_Hthy;
      = #o_TRS02_ST_LMS_Not_Hthy;

NETWORK
TITLE = VC: Write outputs SWS03 (TSS)
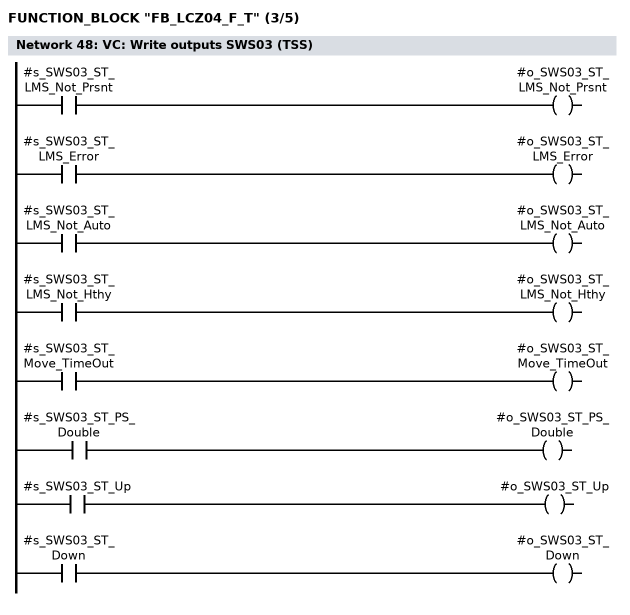
      NOP 0;

// Transfer static values to outputs
      A #s_SWS03_ST_LMS_Not_Prsnt;
      = #o_SWS03_ST_LMS_Not_Prsnt;
      A #s_SWS03_ST_LMS_Error;
      = #o_SWS03_ST_LMS_Error;
      A #s_SWS03_ST_LMS_Not_Auto;
      = #o_SWS03_ST_LMS_Not_Auto;
      A #s_SWS03_ST_LMS_Not_Hthy;
      = #o_SWS03_ST_LMS_Not_Hthy;
      A #s_SWS03_ST_Move_TimeOut;
      = #o_SWS03_ST_Move_TimeOut;
      A #s_SWS03_ST_PS_Double;
      = #o_SWS03_ST_PS_Double;
      A #s_SWS03_ST_Up;
      = #o_SWS03_ST_Up;
      A #s_SWS03_ST_Down;
      = #o_SWS03_ST_Down;

NETWORK
TITLE = VD: Write outputs TRS04 (TTS)
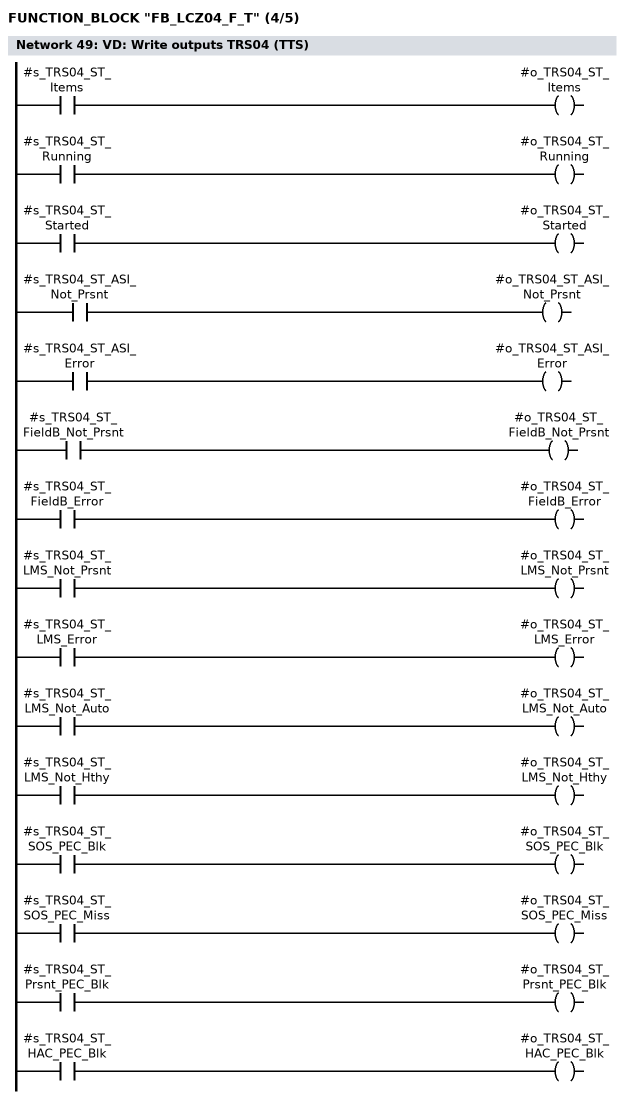
      NOP 0;

// Transfer static values to outputs
      A #s_TRS04_ST_Items;
      = #o_TRS04_ST_Items;
      A #s_TRS04_ST_Running;
      = #o_TRS04_ST_Running;
      A #s_TRS04_ST_Started;
      = #o_TRS04_ST_Started;
      A #s_TRS04_ST_ASI_Not_Prsnt;
      = #o_TRS04_ST_ASI_Not_Prsnt;
      A #s_TRS04_ST_ASI_Error;
      = #o_TRS04_ST_ASI_Error;
      A #s_TRS04_ST_FieldB_Not_Prsnt;
      = #o_TRS04_ST_FieldB_Not_Prsnt;
      A #s_TRS04_ST_FieldB_Error;
      = #o_TRS04_ST_FieldB_Error;
      A #s_TRS04_ST_LMS_Not_Prsnt;
      = #o_TRS04_ST_LMS_Not_Prsnt;
      A #s_TRS04_ST_LMS_Error;
      = #o_TRS04_ST_LMS_Error;
      A #s_TRS04_ST_LMS_Not_Auto;
      = #o_TRS04_ST_LMS_Not_Auto;
      A #s_TRS04_ST_LMS_Not_Hthy;
      = #o_TRS04_ST_LMS_Not_Hthy;
      A #s_TRS04_ST_SOS_PEC_Blk;
      = #o_TRS04_ST_SOS_PEC_Blk;
      A #s_TRS04_ST_SOS_PEC_Miss;
      = #o_TRS04_ST_SOS_PEC_Miss;
      A #s_TRS04_ST_Prsnt_PEC_Blk;
      = #o_TRS04_ST_Prsnt_PEC_Blk;
      A #s_TRS04_ST_HAC_PEC_Blk;
      = #o_TRS04_ST_HAC_PEC_Blk;

NETWORK
TITLE = VE: Write outputs MSO99
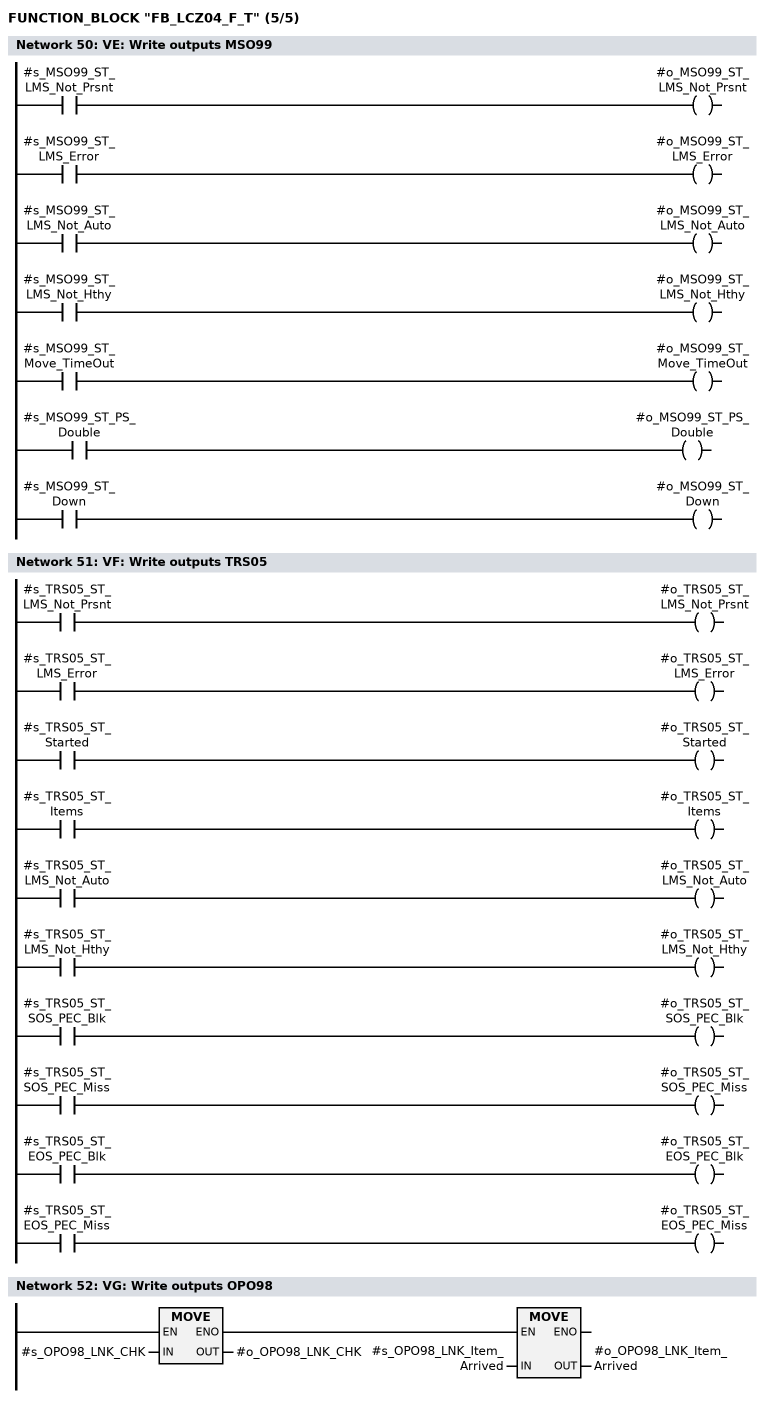
      NOP 0;

// Transfer static values to outputs
      A #s_MSO99_ST_LMS_Not_Prsnt;
      = #o_MSO99_ST_LMS_Not_Prsnt;
      A #s_MSO99_ST_LMS_Error;
      = #o_MSO99_ST_LMS_Error;
      A #s_MSO99_ST_LMS_Not_Auto;
      = #o_MSO99_ST_LMS_Not_Auto;
      A #s_MSO99_ST_LMS_Not_Hthy;
      = #o_MSO99_ST_LMS_Not_Hthy;
      A #s_MSO99_ST_Move_TimeOut;
      = #o_MSO99_ST_Move_TimeOut;
      A #s_MSO99_ST_PS_Double;
      = #o_MSO99_ST_PS_Double;
      A #s_MSO99_ST_Down;
      = #o_MSO99_ST_Down;

NETWORK
TITLE = VF: Write outputs TRS05
      NOP 0;

// Transfer static values to outputs
      A #s_TRS05_ST_LMS_Not_Prsnt;
      = #o_TRS05_ST_LMS_Not_Prsnt;
      A #s_TRS05_ST_LMS_Error;
      = #o_TRS05_ST_LMS_Error;
      A #s_TRS05_ST_Started;
      = #o_TRS05_ST_Started;
      A #s_TRS05_ST_Items;
      = #o_TRS05_ST_Items;
      A #s_TRS05_ST_LMS_Not_Auto;
      = #o_TRS05_ST_LMS_Not_Auto;
      A #s_TRS05_ST_LMS_Not_Hthy;
      = #o_TRS05_ST_LMS_Not_Hthy;
      A #s_TRS05_ST_SOS_PEC_Blk;
      = #o_TRS05_ST_SOS_PEC_Blk;
      A #s_TRS05_ST_SOS_PEC_Miss;
      = #o_TRS05_ST_SOS_PEC_Miss;
      A #s_TRS05_ST_EOS_PEC_Blk;
      = #o_TRS05_ST_EOS_PEC_Blk;
      A #s_TRS05_ST_EOS_PEC_Miss;
      = #o_TRS05_ST_EOS_PEC_Miss;

NETWORK
TITLE = VG: Write outputs OPO98
      NOP 0;

      L #s_OPO98_LNK_CHK;
      T #o_OPO98_LNK_CHK;

      L #s_OPO98_LNK_Item_Arrived;
      T #o_OPO98_LNK_Item_Arrived;

END_FUNCTION_BLOCK

